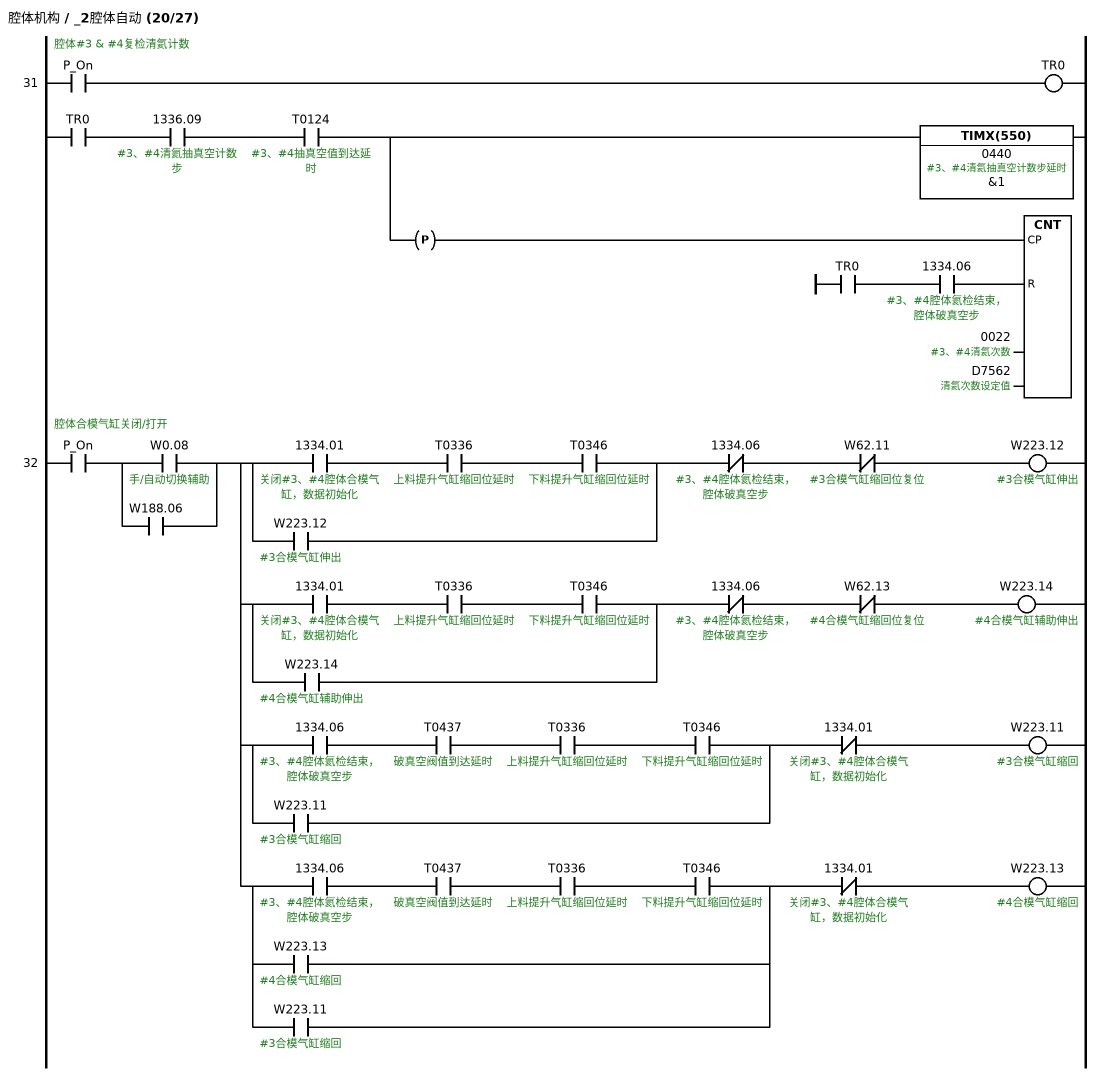
; [picture p288: 腔体机构 / _2腔体自动, rungs 31-32]
; rung 31: 腔体#3 & #4复检清氦计数
LD P_On
OUT TR0
AND 1336.09  ; #3、#4清氦抽真空计数步
AND T0124  ; #3、#4抽真空值到达延时
TIMX(550) 0440 &1  ; #3、#4清氦抽真空计数步延时
UP(521)
LD TR0
AND 1334.06  ; #3、#4腔体氦检结束，腔体破真空步
CNT 0022 D7562  ; 清氦次数设定值, #3、#4清氦次数
; rung 32: 腔体合模气缸关闭/打开
LD P_On
LD W0.08  ; 手/自动切换辅助
OR W188.06
ANDLD
OUT TR0
LD 1334.01  ; 关闭#3、#4腔体合模气缸，数据初始化
AND T0336  ; 上料提升气缸缩回位延时
AND T0346  ; 下料提升气缸缩回位延时
OR W223.12  ; #3合模气缸伸出
ANDLD
ANDNOT 1334.06  ; #3、#4腔体氦检结束，腔体破真空步
ANDNOT W62.11  ; #3合模气缸缩回位复位
OUT W223.12  ; #3合模气缸伸出
LD TR0
LD 1334.01  ; 关闭#3、#4腔体合模气缸，数据初始化
AND T0336  ; 上料提升气缸缩回位延时
AND T0346  ; 下料提升气缸缩回位延时
OR W223.14  ; #4合模气缸辅助伸出
ANDLD
ANDNOT 1334.06  ; #3、#4腔体氦检结束，腔体破真空步
ANDNOT W62.13  ; #4合模气缸缩回位复位
OUT W223.14  ; #4合模气缸辅助伸出
LD TR0
LD 1334.06  ; #3、#4腔体氦检结束，腔体破真空步
AND T0437  ; 破真空阀值到达延时
AND T0336  ; 上料提升气缸缩回位延时
AND T0346  ; 下料提升气缸缩回位延时
OR W223.11  ; #3合模气缸缩回
ANDLD
ANDNOT 1334.01  ; 关闭#3、#4腔体合模气缸，数据初始化
OUT W223.11  ; #3合模气缸缩回
LD TR0
LD 1334.06  ; #3、#4腔体氦检结束，腔体破真空步
AND T0437  ; 破真空阀值到达延时
AND T0336  ; 上料提升气缸缩回位延时
AND T0346  ; 下料提升气缸缩回位延时
LD W223.13  ; #4合模气缸缩回
OR W223.11  ; #3合模气缸缩回
ORLD
ANDLD
ANDNOT 1334.01  ; 关闭#3、#4腔体合模气缸，数据初始化
OUT W223.13  ; #4合模气缸缩回

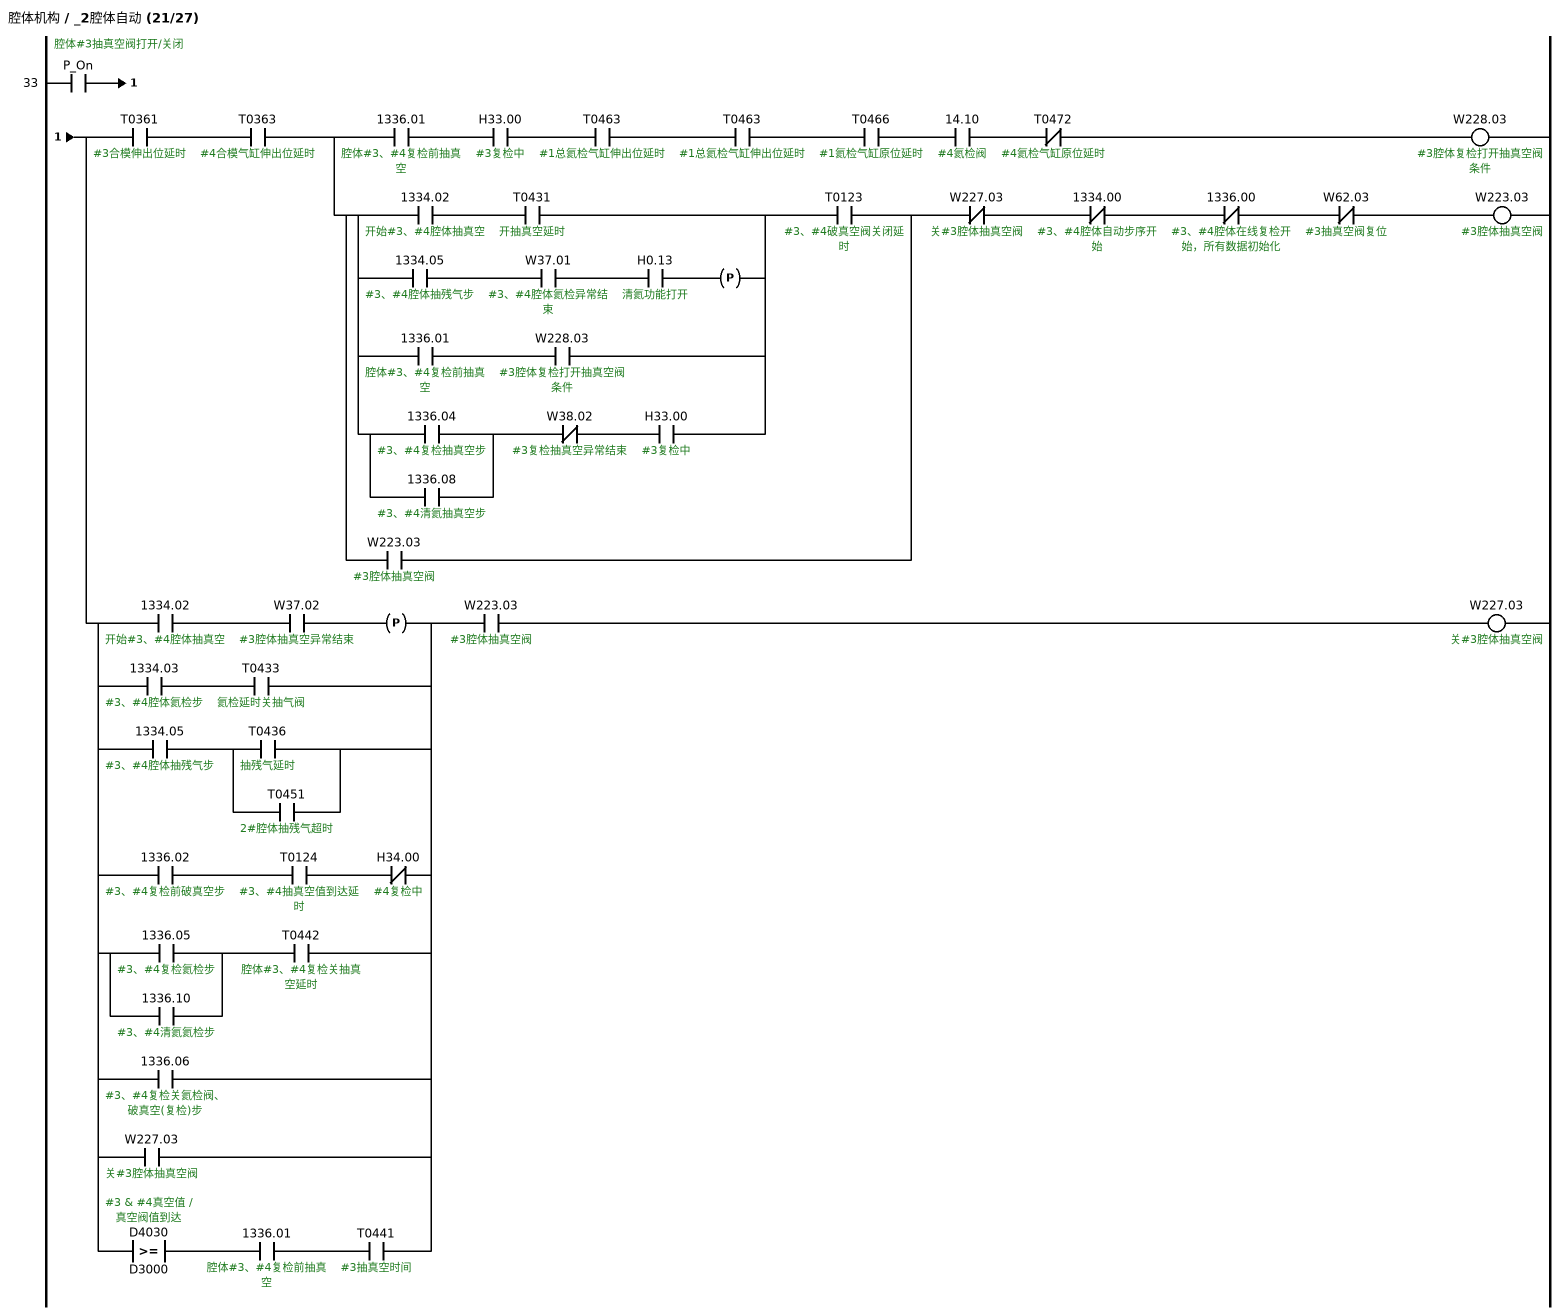
; rung 33: 腔体#3抽真空阀打开/关闭
LD P_On
OUT TR0
AND T0361  ; #3合模伸出位延时
AND T0363  ; #4合模气缸伸出位延时
OUT TR1
AND 1336.01  ; 腔体#3、#4复检前抽真空
AND H33.00  ; #3复检中
AND T0463  ; #1总氦检气缸伸出位延时
AND T0463  ; #1总氦检气缸伸出位延时
AND T0466  ; #1氦检气缸原位延时
AND 14.10  ; #4氦检阀
ANDNOT T0472  ; #4氦检气缸原位延时
OUT W228.03  ; #3腔体复检打开抽真空阀条件
LD TR1
LD 1334.02  ; 开始#3、#4腔体抽真空
AND T0431  ; 开抽真空延时
LD 1334.05  ; #3、#4腔体抽残气步
AND W37.01  ; #3、#4腔体氦检异常结束
AND H0.13  ; 清氦功能打开
UP(521)
ORLD
LD 1336.01  ; 腔体#3、#4复检前抽真空
AND W228.03  ; #3腔体复检打开抽真空阀条件
ORLD
LD 1336.04  ; #3、#4复检抽真空步
OR 1336.08  ; #3、#4清氦抽真空步
ANDNOT W38.02  ; #3复检抽真空异常结束
AND H33.00  ; #3复检中
ORLD
AND T0123  ; #3、#4破真空阀关闭延时
OR W223.03  ; #3腔体抽真空阀
ANDLD
ANDNOT W227.03  ; 关#3腔体抽真空阀
ANDNOT 1334.00  ; #3、#4腔体自动步序开始
ANDNOT 1336.00  ; #3、#4腔体在线复检开始，所有数据初始化
ANDNOT W62.03  ; #3抽真空阀复位
OUT W223.03  ; #3腔体抽真空阀
LD TR0
LD 1334.02  ; 开始#3、#4腔体抽真空
AND W37.02  ; #3腔体抽真空异常结束
UP(521)
LD 1334.03  ; #3、#4腔体氦检步
AND T0433  ; 氦检延时关抽气阀
ORLD
LD 1334.05  ; #3、#4腔体抽残气步
LD T0436  ; 抽残气延时
OR T0451  ; 2#腔体抽残气超时
ANDLD
ORLD
LD 1336.02  ; #3、#4复检前破真空步
AND T0124  ; #3、#4抽真空值到达延时
ANDNOT H34.00  ; #4复检中
ORLD
LD 1336.05  ; #3、#4复检氦检步
OR 1336.10  ; #3、#4清氦氦检步
AND T0442  ; 腔体#3、#4复检关抽真空延时
ORLD
OR 1336.06  ; #3、#4复检关氦检阀、破真空(复检)步
OR W227.03  ; 关#3腔体抽真空阀
LD>=F(334) D4030 D3000  ; #3 & #4真空值, 真空阀值到达
AND 1336.01  ; 腔体#3、#4复检前抽真空
AND T0441  ; #3抽真空时间
ORLD
ANDLD
AND W223.03  ; #3腔体抽真空阀
OUT W227.03  ; 关#3腔体抽真空阀

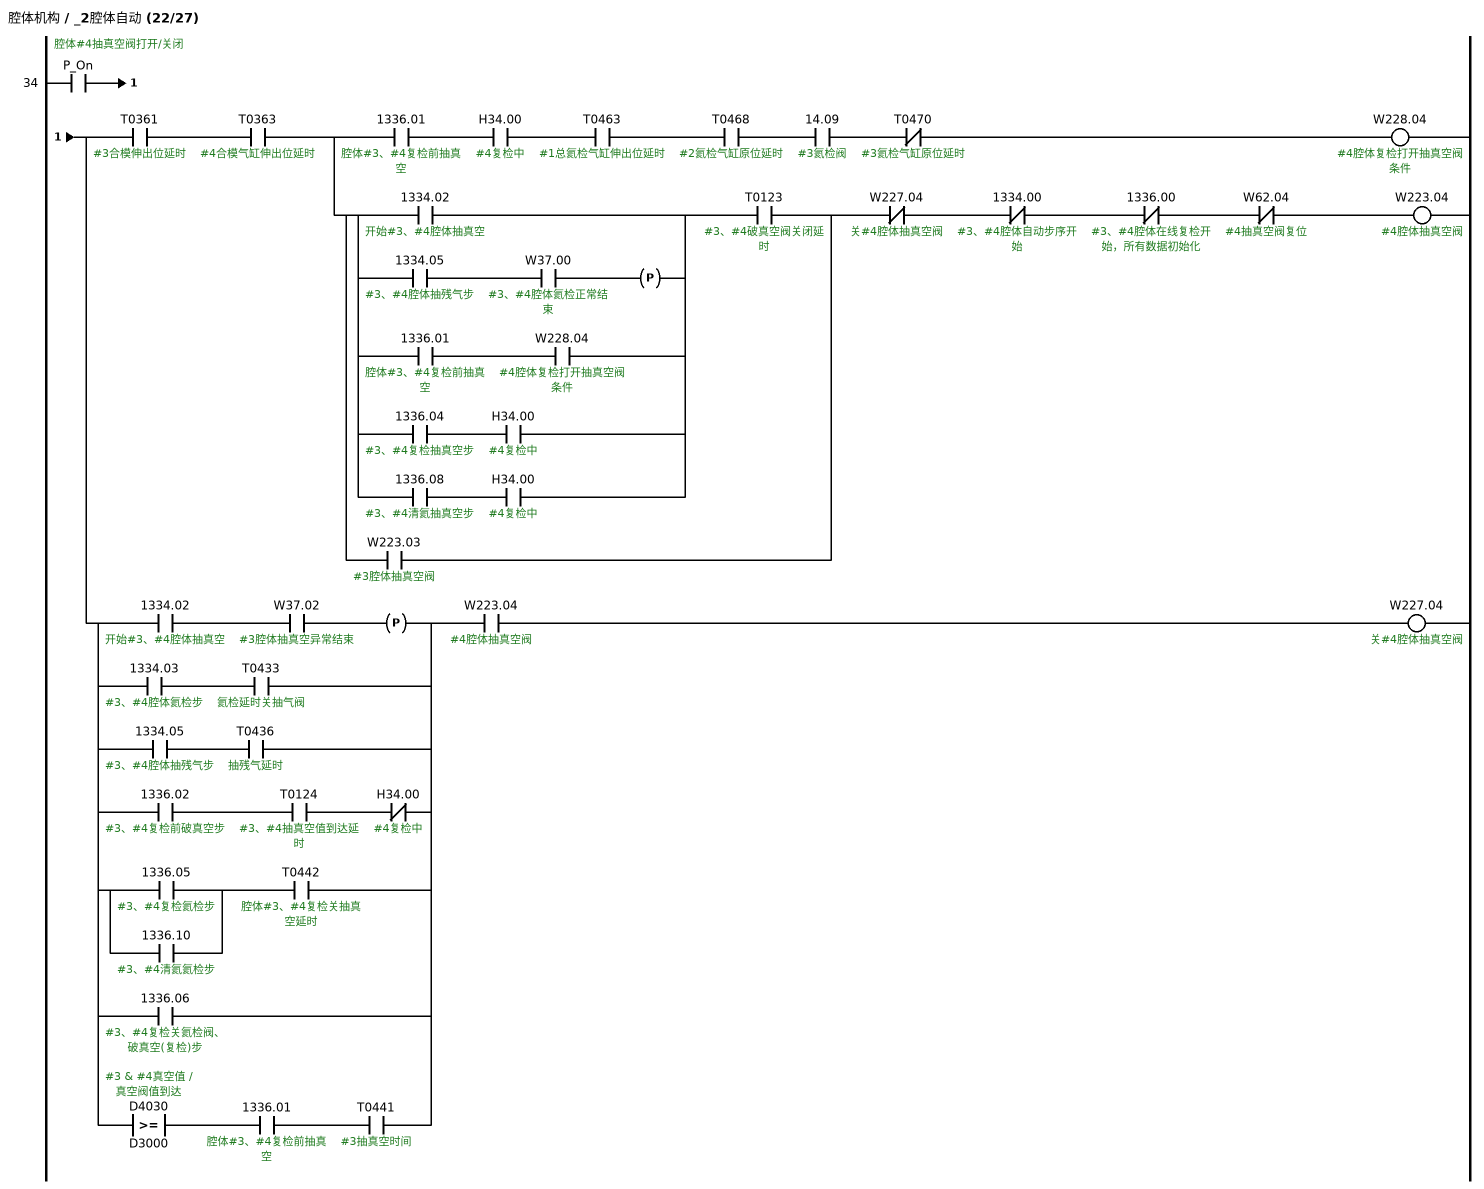
; rung 34: 腔体#4抽真空阀打开/关闭
LD P_On
OUT TR0
AND T0361  ; #3合模伸出位延时
AND T0363  ; #4合模气缸伸出位延时
OUT TR1
AND 1336.01  ; 腔体#3、#4复检前抽真空
AND H34.00  ; #4复检中
AND T0463  ; #1总氦检气缸伸出位延时
AND T0468  ; #2氦检气缸原位延时
AND 14.09  ; #3氦检阀
ANDNOT T0470  ; #3氦检气缸原位延时
OUT W228.04  ; #4腔体复检打开抽真空阀条件
LD TR1
LD 1334.02  ; 开始#3、#4腔体抽真空
LD 1334.05  ; #3、#4腔体抽残气步
AND W37.00  ; #3、#4腔体氦检正常结束
UP(521)
ORLD
LD 1336.01  ; 腔体#3、#4复检前抽真空
AND W228.04  ; #4腔体复检打开抽真空阀条件
ORLD
LD 1336.04  ; #3、#4复检抽真空步
AND H34.00  ; #4复检中
ORLD
LD 1336.08  ; #3、#4清氦抽真空步
AND H34.00  ; #4复检中
ORLD
AND T0123  ; #3、#4破真空阀关闭延时
OR W223.03  ; #3腔体抽真空阀
ANDLD
ANDNOT W227.04  ; 关#4腔体抽真空阀
ANDNOT 1334.00  ; #3、#4腔体自动步序开始
ANDNOT 1336.00  ; #3、#4腔体在线复检开始，所有数据初始化
ANDNOT W62.04  ; #4抽真空阀复位
OUT W223.04  ; #4腔体抽真空阀
LD TR0
LD 1334.02  ; 开始#3、#4腔体抽真空
AND W37.02  ; #3腔体抽真空异常结束
UP(521)
LD 1334.03  ; #3、#4腔体氦检步
AND T0433  ; 氦检延时关抽气阀
ORLD
LD 1334.05  ; #3、#4腔体抽残气步
AND T0436  ; 抽残气延时
ORLD
LD 1336.02  ; #3、#4复检前破真空步
AND T0124  ; #3、#4抽真空值到达延时
ANDNOT H34.00  ; #4复检中
ORLD
LD 1336.05  ; #3、#4复检氦检步
OR 1336.10  ; #3、#4清氦氦检步
AND T0442  ; 腔体#3、#4复检关抽真空延时
ORLD
OR 1336.06  ; #3、#4复检关氦检阀、破真空(复检)步
LD>=F(334) D4030 D3000  ; #3 & #4真空值, 真空阀值到达
AND 1336.01  ; 腔体#3、#4复检前抽真空
AND T0441  ; #3抽真空时间
ORLD
ANDLD
AND W223.04  ; #4腔体抽真空阀
OUT W227.04  ; 关#4腔体抽真空阀

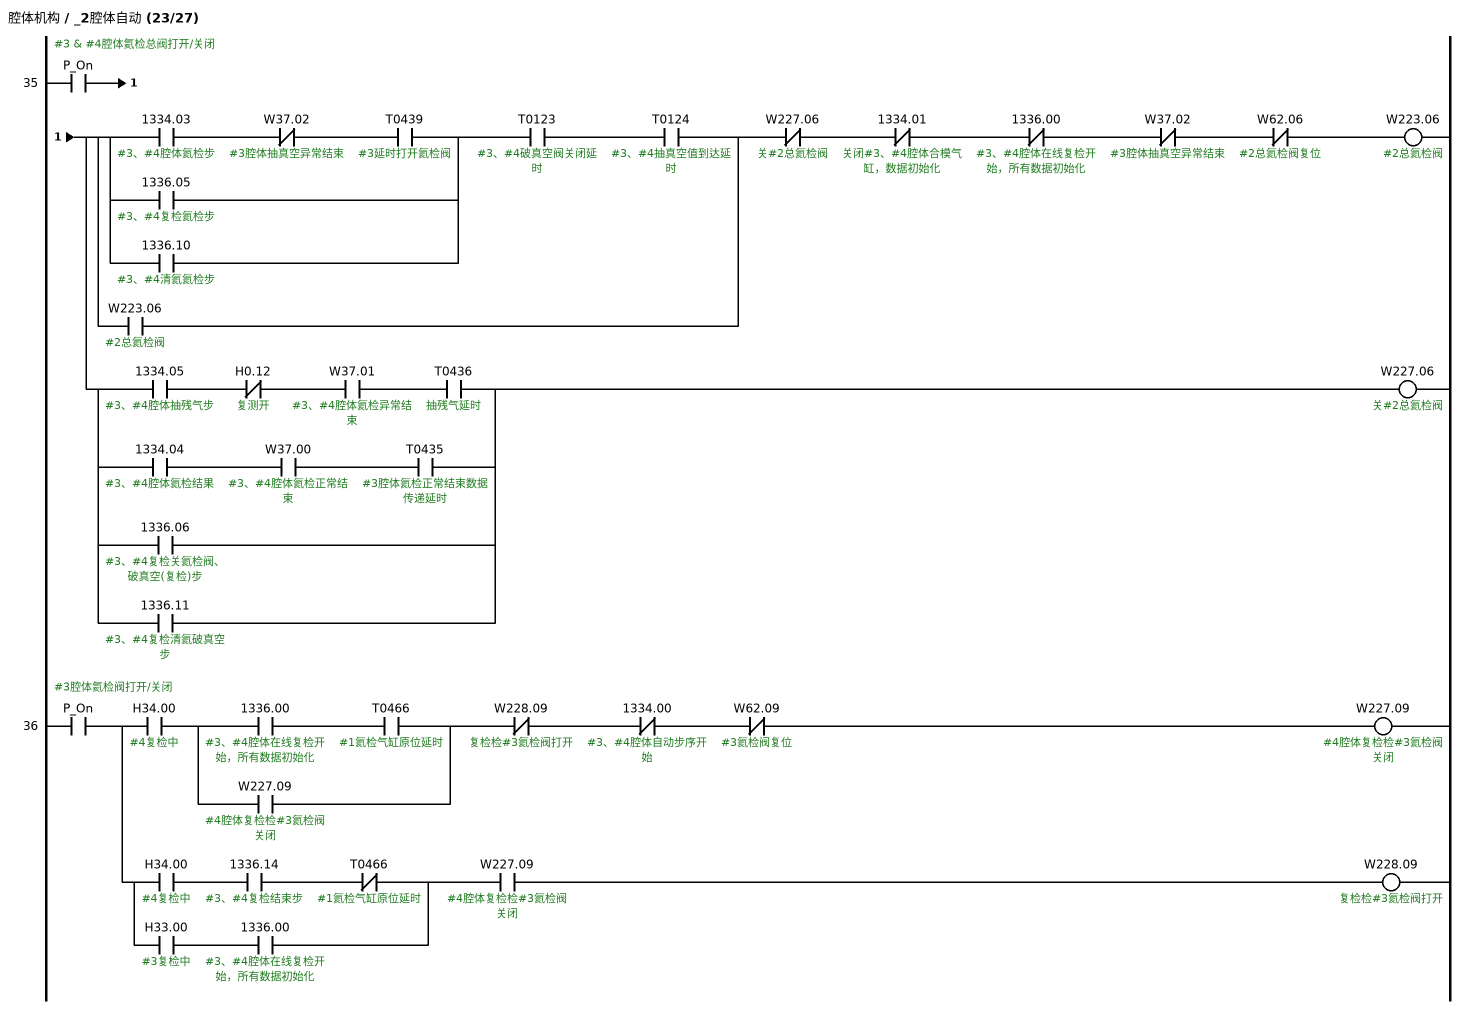
; rung 35: #3 & #4腔体氦检总阀打开/关闭
LD P_On
OUT TR0
LD 1334.03  ; #3、#4腔体氦检步
ANDNOT W37.02  ; #3腔体抽真空异常结束
AND T0439  ; #3延时打开氦检阀
OR 1336.05  ; #3、#4复检氦检步
OR 1336.10  ; #3、#4清氦氦检步
AND T0123  ; #3、#4破真空阀关闭延时
AND T0124  ; #3、#4抽真空值到达延时
OR W223.06  ; #2总氦检阀
ANDLD
ANDNOT W227.06  ; 关#2总氦检阀
ANDNOT 1334.01  ; 关闭#3、#4腔体合模气缸，数据初始化
ANDNOT 1336.00  ; #3、#4腔体在线复检开始，所有数据初始化
ANDNOT W37.02  ; #3腔体抽真空异常结束
ANDNOT W62.06  ; #2总氦检阀复位
OUT W223.06  ; #2总氦检阀
LD TR0
LD 1334.05  ; #3、#4腔体抽残气步
ANDNOT H0.12  ; 复测开
AND W37.01  ; #3、#4腔体氦检异常结束
AND T0436  ; 抽残气延时
LD 1334.04  ; #3、#4腔体氦检结果
AND W37.00  ; #3、#4腔体氦检正常结束
AND T0435  ; #3腔体氦检正常结束数据传递延时
ORLD
OR 1336.06  ; #3、#4复检关氦检阀、破真空(复检)步
OR 1336.11  ; #3、#4复检清氦破真空步
ANDLD
OUT W227.06  ; 关#2总氦检阀
; rung 36: #3腔体氦检阀打开/关闭
LD P_On
OUT TR0
AND H34.00  ; #4复检中
LD 1336.00  ; #3、#4腔体在线复检开始，所有数据初始化
AND T0466  ; #1氦检气缸原位延时
OR W227.09  ; #4腔体复检检#3氦检阀关闭
ANDLD
ANDNOT W228.09  ; 复检检#3氦检阀打开
ANDNOT 1334.00  ; #3、#4腔体自动步序开始
ANDNOT W62.09  ; #3氦检阀复位
OUT W227.09  ; #4腔体复检检#3氦检阀关闭
LD TR0
LD H34.00  ; #4复检中
AND 1336.14  ; #3、#4复检结束步
ANDNOT T0466  ; #1氦检气缸原位延时
LD H33.00  ; #3复检中
AND 1336.00  ; #3、#4腔体在线复检开始，所有数据初始化
ORLD
ANDLD
AND W227.09  ; #4腔体复检检#3氦检阀关闭
OUT W228.09  ; 复检检#3氦检阀打开

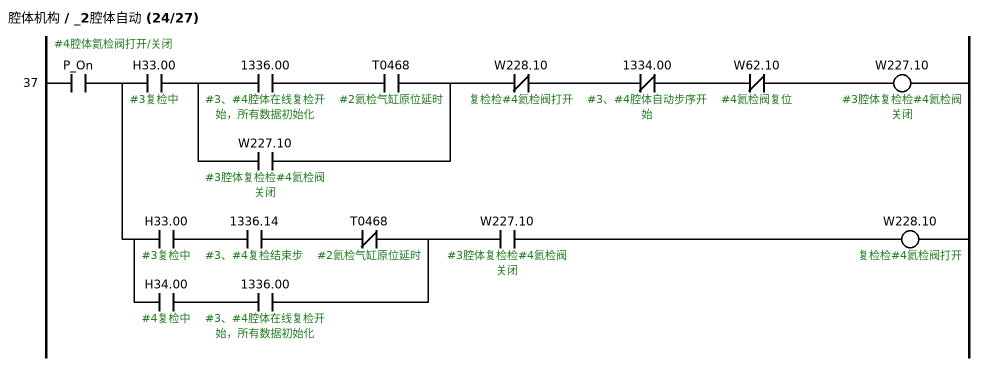
; rung 37: #4腔体氦检阀打开/关闭
LD P_On
OUT TR0
AND H33.00  ; #3复检中
LD 1336.00  ; #3、#4腔体在线复检开始，所有数据初始化
AND T0468  ; #2氦检气缸原位延时
OR W227.10  ; #3腔体复检检#4氦检阀关闭
ANDLD
ANDNOT W228.10  ; 复检检#4氦检阀打开
ANDNOT 1334.00  ; #3、#4腔体自动步序开始
ANDNOT W62.10  ; #4氦检阀复位
OUT W227.10  ; #3腔体复检检#4氦检阀关闭
LD TR0
LD H33.00  ; #3复检中
AND 1336.14  ; #3、#4复检结束步
ANDNOT T0468  ; #2氦检气缸原位延时
LD H34.00  ; #4复检中
AND 1336.00  ; #3、#4腔体在线复检开始，所有数据初始化
ORLD
ANDLD
AND W227.10  ; #3腔体复检检#4氦检阀关闭
OUT W228.10  ; 复检检#4氦检阀打开

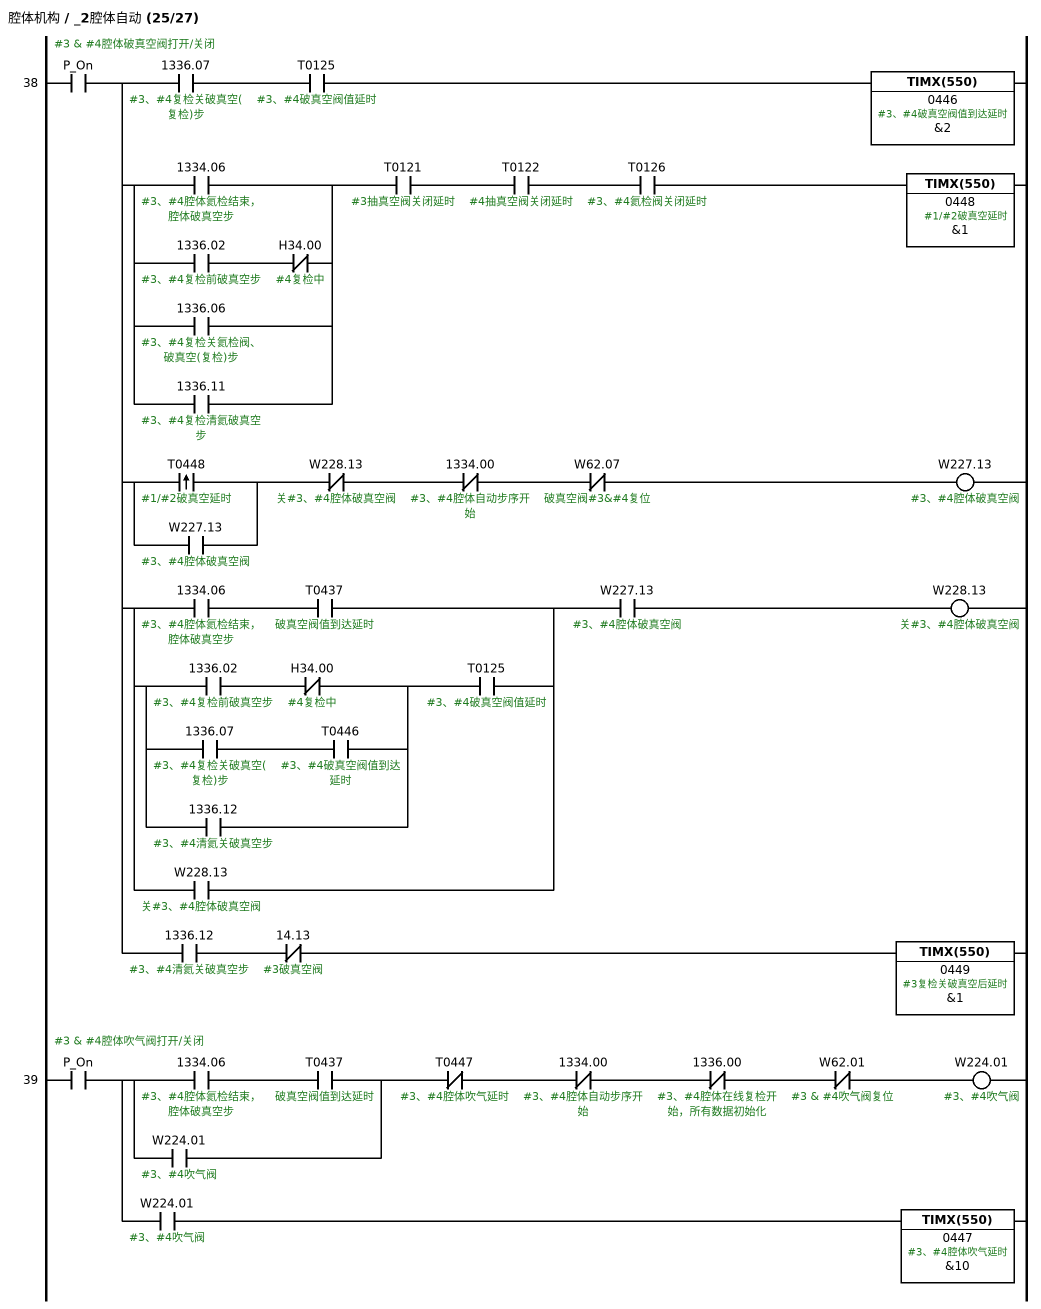
; rung 38: #3 & #4腔体破真空阀打开/关闭
LD P_On
OUT TR0
AND 1336.07  ; #3、#4复检关破真空(复检)步
AND T0125  ; #3、#4破真空阀值延时
TIMX(550) 0446 &2  ; #3、#4破真空阀值到达延时
LD TR0
LD 1334.06  ; #3、#4腔体氦检结束，腔体破真空步
LD 1336.02  ; #3、#4复检前破真空步
ANDNOT H34.00  ; #4复检中
ORLD
OR 1336.06  ; #3、#4复检关氦检阀、破真空(复检)步
OR 1336.11  ; #3、#4复检清氦破真空步
ANDLD
AND T0121  ; #3抽真空阀关闭延时
AND T0122  ; #4抽真空阀关闭延时
AND T0126  ; #3、#4氦检阀关闭延时
TIMX(550) 0448 &1  ; #1/#2破真空延时
LD TR0
@LD T0448  ; #1/#2破真空延时
OR W227.13  ; #3、#4腔体破真空阀
ANDLD
ANDNOT W228.13  ; 关#3、#4腔体破真空阀
ANDNOT 1334.00  ; #3、#4腔体自动步序开始
ANDNOT W62.07  ; 破真空阀#3&#4复位
OUT W227.13  ; #3、#4腔体破真空阀
LD TR0
LD 1334.06  ; #3、#4腔体氦检结束，腔体破真空步
AND T0437  ; 破真空阀值到达延时
LD 1336.02  ; #3、#4复检前破真空步
ANDNOT H34.00  ; #4复检中
LD 1336.07  ; #3、#4复检关破真空(复检)步
AND T0446  ; #3、#4破真空阀值到达延时
ORLD
OR 1336.12  ; #3、#4清氦关破真空步
AND T0125  ; #3、#4破真空阀值延时
ORLD
OR W228.13  ; 关#3、#4腔体破真空阀
ANDLD
AND W227.13  ; #3、#4腔体破真空阀
OUT W228.13  ; 关#3、#4腔体破真空阀
LD TR0
AND 1336.12  ; #3、#4清氦关破真空步
ANDNOT 14.13  ; #3破真空阀
TIMX(550) 0449 &1  ; #3复检关破真空后延时
; rung 39: #3 & #4腔体吹气阀打开/关闭
LD P_On
OUT TR0
LD 1334.06  ; #3、#4腔体氦检结束，腔体破真空步
AND T0437  ; 破真空阀值到达延时
OR W224.01  ; #3、#4吹气阀
ANDLD
ANDNOT T0447  ; #3、#4腔体吹气延时
ANDNOT 1334.00  ; #3、#4腔体自动步序开始
ANDNOT 1336.00  ; #3、#4腔体在线复检开始，所有数据初始化
ANDNOT W62.01  ; #3 & #4吹气阀复位
OUT W224.01  ; #3、#4吹气阀
LD TR0
AND W224.01  ; #3、#4吹气阀
TIMX(550) 0447 &10  ; #3、#4腔体吹气延时

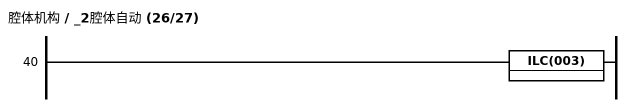
; rung 40
ILC(003)

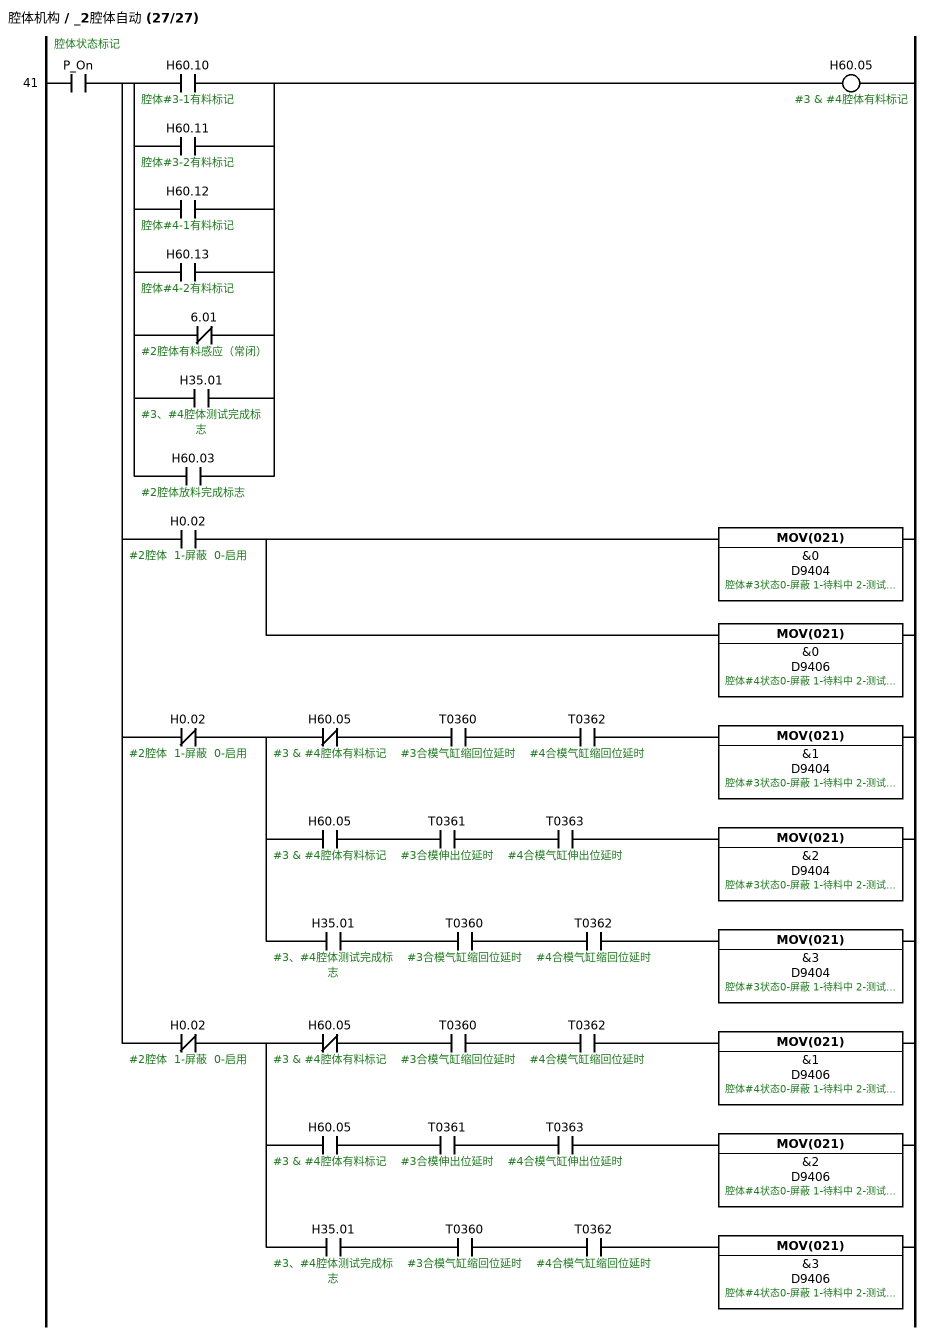
; rung 41: 腔体状态标记
LD P_On
OUT TR0
LD H60.10  ; 腔体#3-1有料标记
OR H60.11  ; 腔体#3-2有料标记
OR H60.12  ; 腔体#4-1有料标记
OR H60.13  ; 腔体#4-2有料标记
ORNOT 6.01  ; #2腔体有料感应（常闭）
OR H35.01  ; #3、#4腔体测试完成标志
OR H60.03  ; #2腔体放料完成标志
ANDLD
OUT H60.05  ; #3 & #4腔体有料标记
LD TR0
AND H0.02  ; #2腔体  1-屏蔽  0-启用
MOV(021) &0 D9404  ; 腔体#3状态0-屏蔽 1-待料中 2-测试中 3-测试完成 4-在线复检
MOV(021) &0 D9406  ; 腔体#4状态0-屏蔽 1-待料中 2-测试中 3-测试完成 4-在线复检
LD TR0
ANDNOT H0.02  ; #2腔体  1-屏蔽  0-启用
OUT TR1
ANDNOT H60.05  ; #3 & #4腔体有料标记
AND T0360  ; #3合模气缸缩回位延时
AND T0362  ; #4合模气缸缩回位延时
MOV(021) &1 D9404  ; 腔体#3状态0-屏蔽 1-待料中 2-测试中 3-测试完成 4-在线复检
LD TR1
AND H60.05  ; #3 & #4腔体有料标记
AND T0361  ; #3合模伸出位延时
AND T0363  ; #4合模气缸伸出位延时
MOV(021) &2 D9404  ; 腔体#3状态0-屏蔽 1-待料中 2-测试中 3-测试完成 4-在线复检
LD TR1
AND H35.01  ; #3、#4腔体测试完成标志
AND T0360  ; #3合模气缸缩回位延时
AND T0362  ; #4合模气缸缩回位延时
MOV(021) &3 D9404  ; 腔体#3状态0-屏蔽 1-待料中 2-测试中 3-测试完成 4-在线复检
LD TR0
ANDNOT H0.02  ; #2腔体  1-屏蔽  0-启用
OUT TR0
ANDNOT H60.05  ; #3 & #4腔体有料标记
AND T0360  ; #3合模气缸缩回位延时
AND T0362  ; #4合模气缸缩回位延时
MOV(021) &1 D9406  ; 腔体#4状态0-屏蔽 1-待料中 2-测试中 3-测试完成 4-在线复检
LD TR0
AND H60.05  ; #3 & #4腔体有料标记
AND T0361  ; #3合模伸出位延时
AND T0363  ; #4合模气缸伸出位延时
MOV(021) &2 D9406  ; 腔体#4状态0-屏蔽 1-待料中 2-测试中 3-测试完成 4-在线复检
LD TR0
AND H35.01  ; #3、#4腔体测试完成标志
AND T0360  ; #3合模气缸缩回位延时
AND T0362  ; #4合模气缸缩回位延时
MOV(021) &3 D9406  ; 腔体#4状态0-屏蔽 1-待料中 2-测试中 3-测试完成 4-在线复检

### Section 腔体机构手动

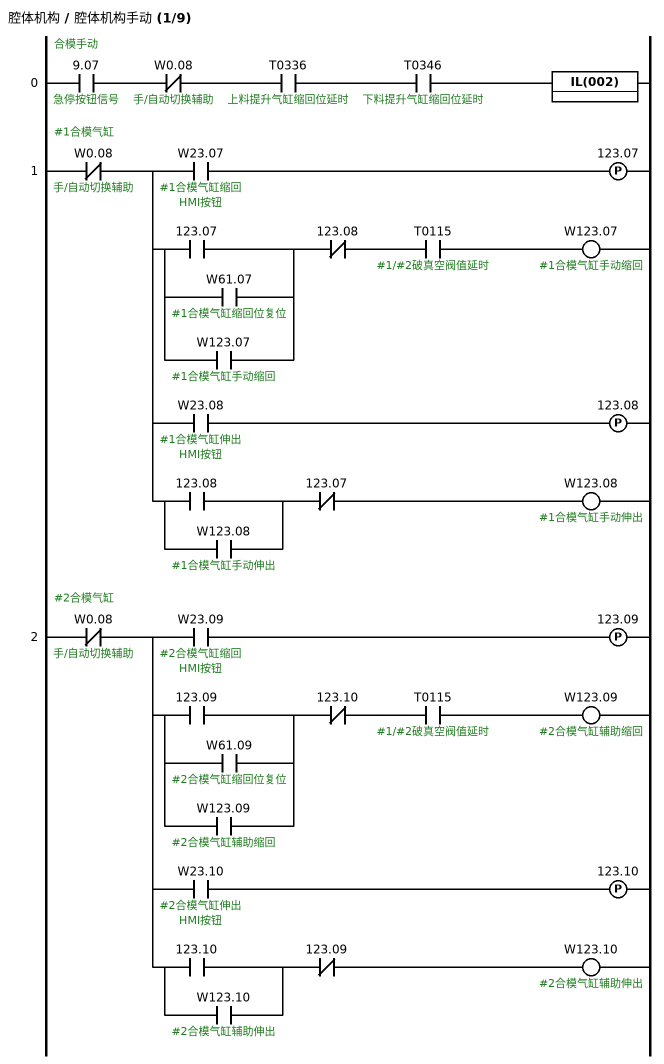
; rung 0: 合模手动
LD 9.07  ; 急停按钮信号
ANDNOT W0.08  ; 手/自动切换辅助
AND T0336  ; 上料提升气缸缩回位延时
AND T0346  ; 下料提升气缸缩回位延时
IL(002)
; rung 1: #1合模气缸
LDNOT W0.08  ; 手/自动切换辅助
OUT TR0
AND W23.07  ; #1合模气缸缩回   HMI按钮
DIFU(013) 123.07
LD TR0
LD 123.07
OR W61.07  ; #1合模气缸缩回位复位
OR W123.07  ; #1合模气缸手动缩回
ANDLD
ANDNOT 123.08
AND T0115  ; #1/#2破真空阀值延时
OUT W123.07  ; #1合模气缸手动缩回
LD TR0
AND W23.08  ; #1合模气缸伸出   HMI按钮
DIFU(013) 123.08
LD TR0
LD 123.08
OR W123.08  ; #1合模气缸手动伸出
ANDLD
ANDNOT 123.07
OUT W123.08  ; #1合模气缸手动伸出
; rung 2: #2合模气缸
LDNOT W0.08  ; 手/自动切换辅助
OUT TR0
AND W23.09  ; #2合模气缸缩回   HMI按钮
DIFU(013) 123.09
LD TR0
LD 123.09
OR W61.09  ; #2合模气缸缩回位复位
OR W123.09  ; #2合模气缸辅助缩回
ANDLD
ANDNOT 123.10
AND T0115  ; #1/#2破真空阀值延时
OUT W123.09  ; #2合模气缸辅助缩回
LD TR0
AND W23.10  ; #2合模气缸伸出   HMI按钮
DIFU(013) 123.10
LD TR0
LD 123.10
OR W123.10  ; #2合模气缸辅助伸出
ANDLD
ANDNOT 123.09
OUT W123.10  ; #2合模气缸辅助伸出

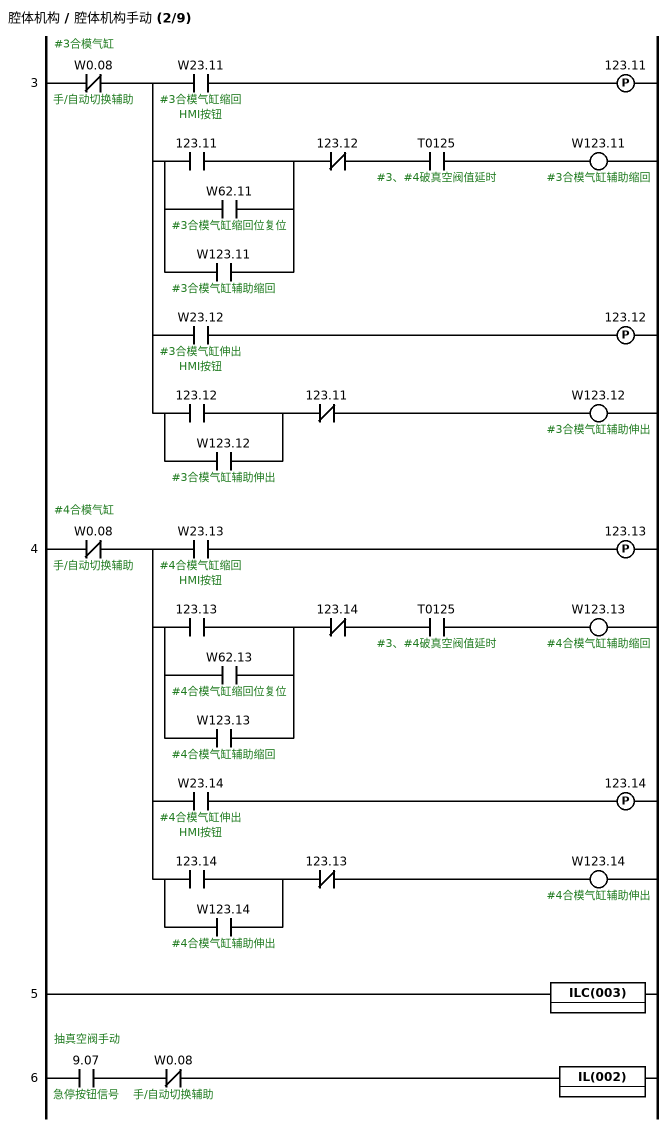
; rung 3: #3合模气缸
LDNOT W0.08  ; 手/自动切换辅助
OUT TR0
AND W23.11  ; #3合模气缸缩回   HMI按钮
DIFU(013) 123.11
LD TR0
LD 123.11
OR W62.11  ; #3合模气缸缩回位复位
OR W123.11  ; #3合模气缸辅助缩回
ANDLD
ANDNOT 123.12
AND T0125  ; #3、#4破真空阀值延时
OUT W123.11  ; #3合模气缸辅助缩回
LD TR0
AND W23.12  ; #3合模气缸伸出   HMI按钮
DIFU(013) 123.12
LD TR0
LD 123.12
OR W123.12  ; #3合模气缸辅助伸出
ANDLD
ANDNOT 123.11
OUT W123.12  ; #3合模气缸辅助伸出
; rung 4: #4合模气缸
LDNOT W0.08  ; 手/自动切换辅助
OUT TR0
AND W23.13  ; #4合模气缸缩回   HMI按钮
DIFU(013) 123.13
LD TR0
LD 123.13
OR W62.13  ; #4合模气缸缩回位复位
OR W123.13  ; #4合模气缸辅助缩回
ANDLD
ANDNOT 123.14
AND T0125  ; #3、#4破真空阀值延时
OUT W123.13  ; #4合模气缸辅助缩回
LD TR0
AND W23.14  ; #4合模气缸伸出   HMI按钮
DIFU(013) 123.14
LD TR0
LD 123.14
OR W123.14  ; #4合模气缸辅助伸出
ANDLD
ANDNOT 123.13
OUT W123.14  ; #4合模气缸辅助伸出
; rung 5
ILC(003)
; rung 6: 抽真空阀手动
LD 9.07  ; 急停按钮信号
ANDNOT W0.08  ; 手/自动切换辅助
IL(002)

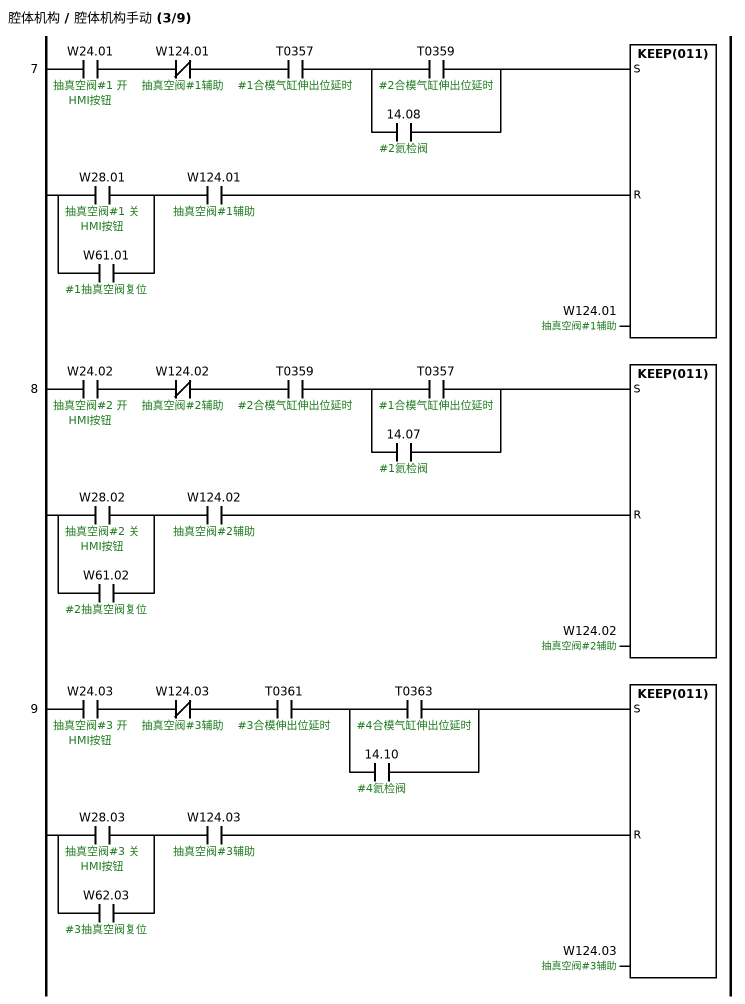
; rung 7
LD W24.01  ; 抽真空阀#1 开    HMI按钮
ANDNOT W124.01  ; 抽真空阀#1辅助
AND T0357  ; #1合模气缸伸出位延时
LD T0359  ; #2合模气缸伸出位延时
OR 14.08  ; #2氦检阀
ANDLD
LD W28.01  ; 抽真空阀#1 关    HMI按钮
OR W61.01  ; #1抽真空阀复位
AND W124.01  ; 抽真空阀#1辅助
KEEP(011) W124.01  ; 抽真空阀#1辅助
; rung 8
LD W24.02  ; 抽真空阀#2 开    HMI按钮
ANDNOT W124.02  ; 抽真空阀#2辅助
AND T0359  ; #2合模气缸伸出位延时
LD T0357  ; #1合模气缸伸出位延时
OR 14.07  ; #1氦检阀
ANDLD
LD W28.02  ; 抽真空阀#2 关    HMI按钮
OR W61.02  ; #2抽真空阀复位
AND W124.02  ; 抽真空阀#2辅助
KEEP(011) W124.02  ; 抽真空阀#2辅助
; rung 9
LD W24.03  ; 抽真空阀#3 开    HMI按钮
ANDNOT W124.03  ; 抽真空阀#3辅助
AND T0361  ; #3合模伸出位延时
LD T0363  ; #4合模气缸伸出位延时
OR 14.10  ; #4氦检阀
ANDLD
LD W28.03  ; 抽真空阀#3 关    HMI按钮
OR W62.03  ; #3抽真空阀复位
AND W124.03  ; 抽真空阀#3辅助
KEEP(011) W124.03  ; 抽真空阀#3辅助

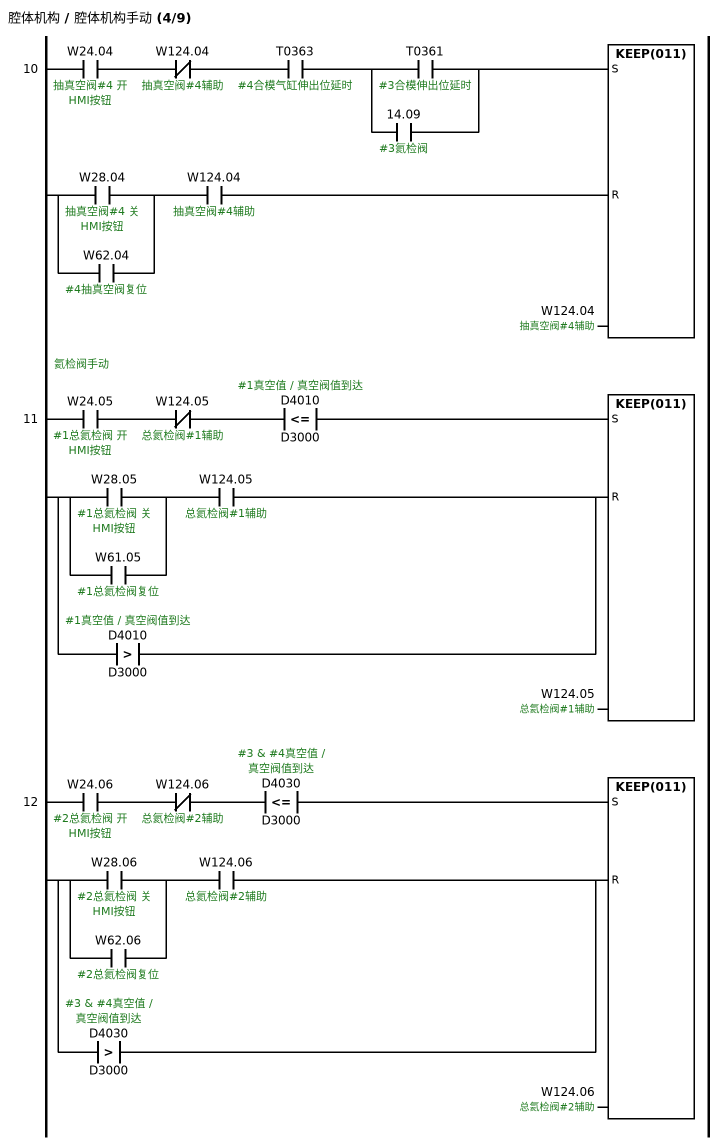
; rung 10
LD W24.04  ; 抽真空阀#4 开    HMI按钮
ANDNOT W124.04  ; 抽真空阀#4辅助
AND T0363  ; #4合模气缸伸出位延时
LD T0361  ; #3合模伸出位延时
OR 14.09  ; #3氦检阀
ANDLD
LD W28.04  ; 抽真空阀#4 关    HMI按钮
OR W62.04  ; #4抽真空阀复位
AND W124.04  ; 抽真空阀#4辅助
KEEP(011) W124.04  ; 抽真空阀#4辅助
; rung 11: 氦检阀手动
LD W24.05  ; #1总氦检阀 开    HMI按钮
ANDNOT W124.05  ; 总氦检阀#1辅助
AND<=F(332) D4010 D3000  ; #1真空值, 真空阀值到达
LD W28.05  ; #1总氦检阀 关    HMI按钮
OR W61.05  ; #1总氦检阀复位
AND W124.05  ; 总氦检阀#1辅助
OR>F(333) D4010 D3000  ; #1真空值, 真空阀值到达
KEEP(011) W124.05  ; 总氦检阀#1辅助
; rung 12
LD W24.06  ; #2总氦检阀 开    HMI按钮
ANDNOT W124.06  ; 总氦检阀#2辅助
AND<=F(332) D4030 D3000  ; #3 & #4真空值, 真空阀值到达
LD W28.06  ; #2总氦检阀 关    HMI按钮
OR W62.06  ; #2总氦检阀复位
AND W124.06  ; 总氦检阀#2辅助
OR>F(333) D4030 D3000  ; #3 & #4真空值, 真空阀值到达
KEEP(011) W124.06  ; 总氦检阀#2辅助

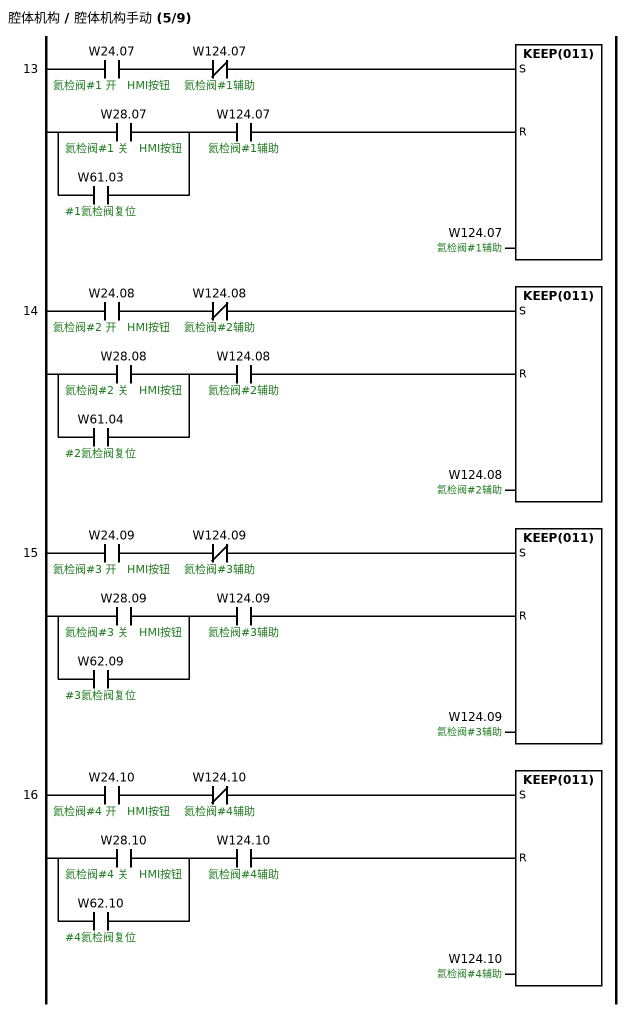
; rung 13
LD W24.07  ; 氦检阀#1 开   HMI按钮
ANDNOT W124.07  ; 氦检阀#1辅助
LD W28.07  ; 氦检阀#1 关   HMI按钮
OR W61.03  ; #1氦检阀复位
AND W124.07  ; 氦检阀#1辅助
KEEP(011) W124.07  ; 氦检阀#1辅助
; rung 14
LD W24.08  ; 氦检阀#2 开   HMI按钮
ANDNOT W124.08  ; 氦检阀#2辅助
LD W28.08  ; 氦检阀#2 关   HMI按钮
OR W61.04  ; #2氦检阀复位
AND W124.08  ; 氦检阀#2辅助
KEEP(011) W124.08  ; 氦检阀#2辅助
; rung 15
LD W24.09  ; 氦检阀#3 开   HMI按钮
ANDNOT W124.09  ; 氦检阀#3辅助
LD W28.09  ; 氦检阀#3 关   HMI按钮
OR W62.09  ; #3氦检阀复位
AND W124.09  ; 氦检阀#3辅助
KEEP(011) W124.09  ; 氦检阀#3辅助
; rung 16
LD W24.10  ; 氦检阀#4 开   HMI按钮
ANDNOT W124.10  ; 氦检阀#4辅助
LD W28.10  ; 氦检阀#4 关   HMI按钮
OR W62.10  ; #4氦检阀复位
AND W124.10  ; 氦检阀#4辅助
KEEP(011) W124.10  ; 氦检阀#4辅助

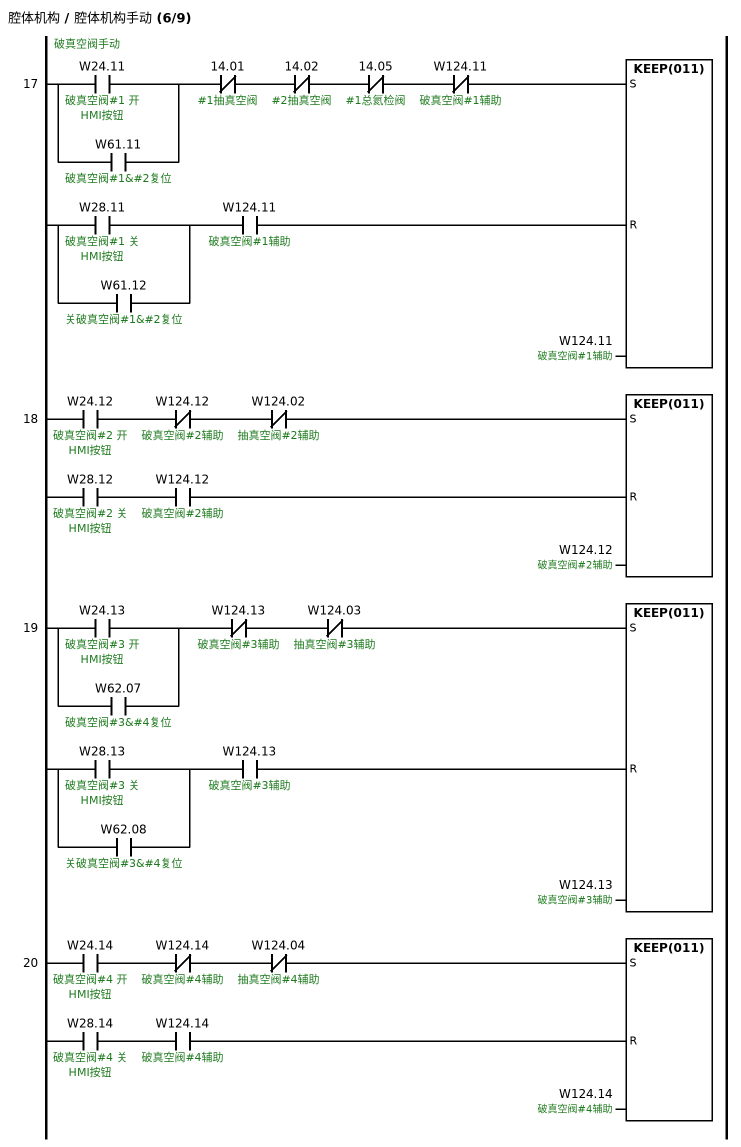
; rung 17: 破真空阀手动
LD W24.11  ; 破真空阀#1 开   HMI按钮
OR W61.11  ; 破真空阀#1&#2复位
ANDNOT 14.01  ; #1抽真空阀
ANDNOT 14.02  ; #2抽真空阀
ANDNOT 14.05  ; #1总氦检阀
ANDNOT W124.11  ; 破真空阀#1辅助
LD W28.11  ; 破真空阀#1 关   HMI按钮
OR W61.12  ; 关破真空阀#1&#2复位
AND W124.11  ; 破真空阀#1辅助
KEEP(011) W124.11  ; 破真空阀#1辅助
; rung 18
LD W24.12  ; 破真空阀#2 开   HMI按钮
ANDNOT W124.12  ; 破真空阀#2辅助
ANDNOT W124.02  ; 抽真空阀#2辅助
LD W28.12  ; 破真空阀#2 关   HMI按钮
AND W124.12  ; 破真空阀#2辅助
KEEP(011) W124.12  ; 破真空阀#2辅助
; rung 19
LD W24.13  ; 破真空阀#3 开   HMI按钮
OR W62.07  ; 破真空阀#3&#4复位
ANDNOT W124.13  ; 破真空阀#3辅助
ANDNOT W124.03  ; 抽真空阀#3辅助
LD W28.13  ; 破真空阀#3 关   HMI按钮
OR W62.08  ; 关破真空阀#3&#4复位
AND W124.13  ; 破真空阀#3辅助
KEEP(011) W124.13  ; 破真空阀#3辅助
; rung 20
LD W24.14  ; 破真空阀#4 开   HMI按钮
ANDNOT W124.14  ; 破真空阀#4辅助
ANDNOT W124.04  ; 抽真空阀#4辅助
LD W28.14  ; 破真空阀#4 关   HMI按钮
AND W124.14  ; 破真空阀#4辅助
KEEP(011) W124.14  ; 破真空阀#4辅助

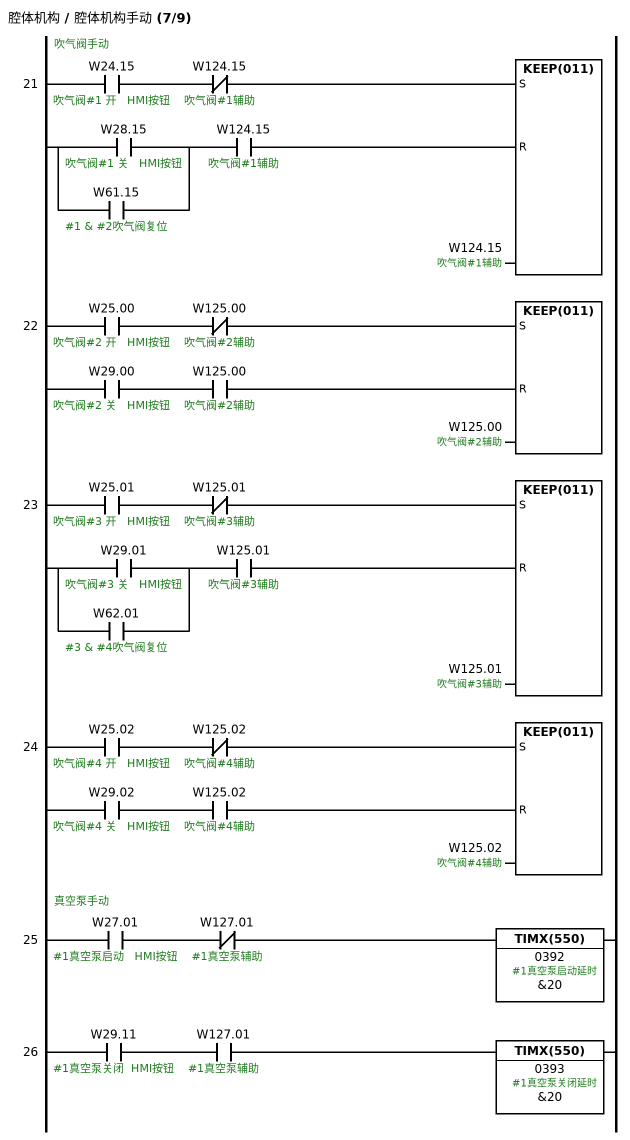
; rung 21: 吹气阀手动
LD W24.15  ; 吹气阀#1 开   HMI按钮
ANDNOT W124.15  ; 吹气阀#1辅助
LD W28.15  ; 吹气阀#1 关   HMI按钮
OR W61.15  ; #1 & #2吹气阀复位
AND W124.15  ; 吹气阀#1辅助
KEEP(011) W124.15  ; 吹气阀#1辅助
; rung 22
LD W25.00  ; 吹气阀#2 开   HMI按钮
ANDNOT W125.00  ; 吹气阀#2辅助
LD W29.00  ; 吹气阀#2 关   HMI按钮
AND W125.00  ; 吹气阀#2辅助
KEEP(011) W125.00  ; 吹气阀#2辅助
; rung 23
LD W25.01  ; 吹气阀#3 开   HMI按钮
ANDNOT W125.01  ; 吹气阀#3辅助
LD W29.01  ; 吹气阀#3 关   HMI按钮
OR W62.01  ; #3 & #4吹气阀复位
AND W125.01  ; 吹气阀#3辅助
KEEP(011) W125.01  ; 吹气阀#3辅助
; rung 24
LD W25.02  ; 吹气阀#4 开   HMI按钮
ANDNOT W125.02  ; 吹气阀#4辅助
LD W29.02  ; 吹气阀#4 关   HMI按钮
AND W125.02  ; 吹气阀#4辅助
KEEP(011) W125.02  ; 吹气阀#4辅助
; rung 25: 真空泵手动
LD W27.01  ; #1真空泵启动   HMI按钮
ANDNOT W127.01  ; #1真空泵辅助
TIMX(550) 0392 &20  ; #1真空泵启动延时
; rung 26
LD W29.11  ; #1真空泵关闭  HMI按钮
AND W127.01  ; #1真空泵辅助
TIMX(550) 0393 &20  ; #1真空泵关闭延时

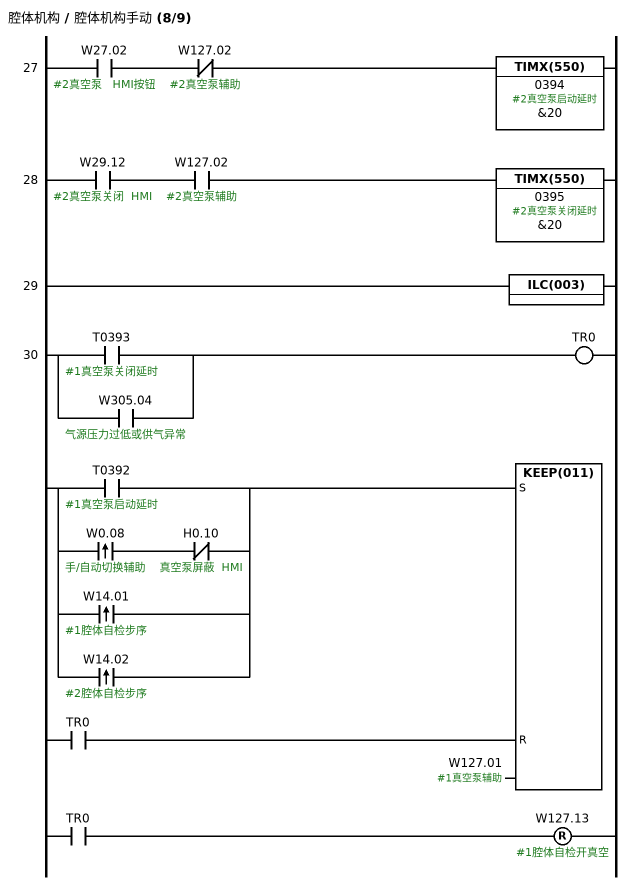
; rung 27
LD W27.02  ; #2真空泵   HMI按钮
ANDNOT W127.02  ; #2真空泵辅助
TIMX(550) 0394 &20  ; #2真空泵启动延时
; rung 28
LD W29.12  ; #2真空泵关闭  HMI
AND W127.02  ; #2真空泵辅助
TIMX(550) 0395 &20  ; #2真空泵关闭延时
; rung 29
ILC(003)
; rung 30
LD T0392  ; #1真空泵启动延时
@LD W0.08  ; 手/自动切换辅助
ANDNOT H0.10  ; 真空泵屏蔽  HMI
ORLD
@OR W14.01  ; #1腔体自检步序
@OR W14.02  ; #2腔体自检步序
LD T0393  ; #1真空泵关闭延时
OR W305.04  ; 气源压力过低或供气异常
OUT TR0
KEEP(011) W127.01  ; #1真空泵辅助
LD TR0
RSET W127.13  ; #1腔体自检开真空

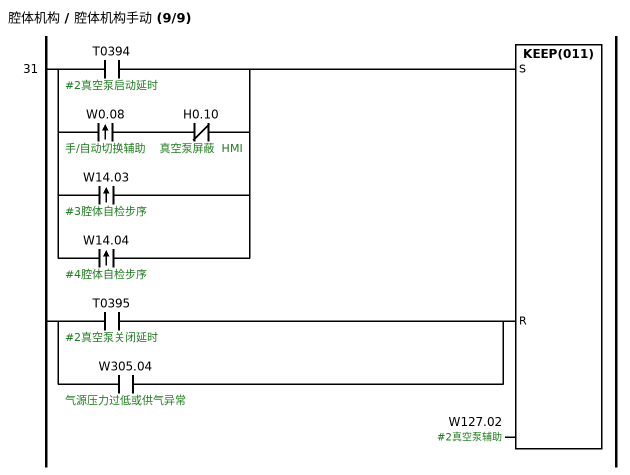
; rung 31
LD T0394  ; #2真空泵启动延时
@LD W0.08  ; 手/自动切换辅助
ANDNOT H0.10  ; 真空泵屏蔽  HMI
ORLD
@OR W14.03  ; #3腔体自检步序
@OR W14.04  ; #4腔体自检步序
LD T0395  ; #2真空泵关闭延时
OR W305.04  ; 气源压力过低或供气异常
KEEP(011) W127.02  ; #2真空泵辅助

### Section _1腔体自检

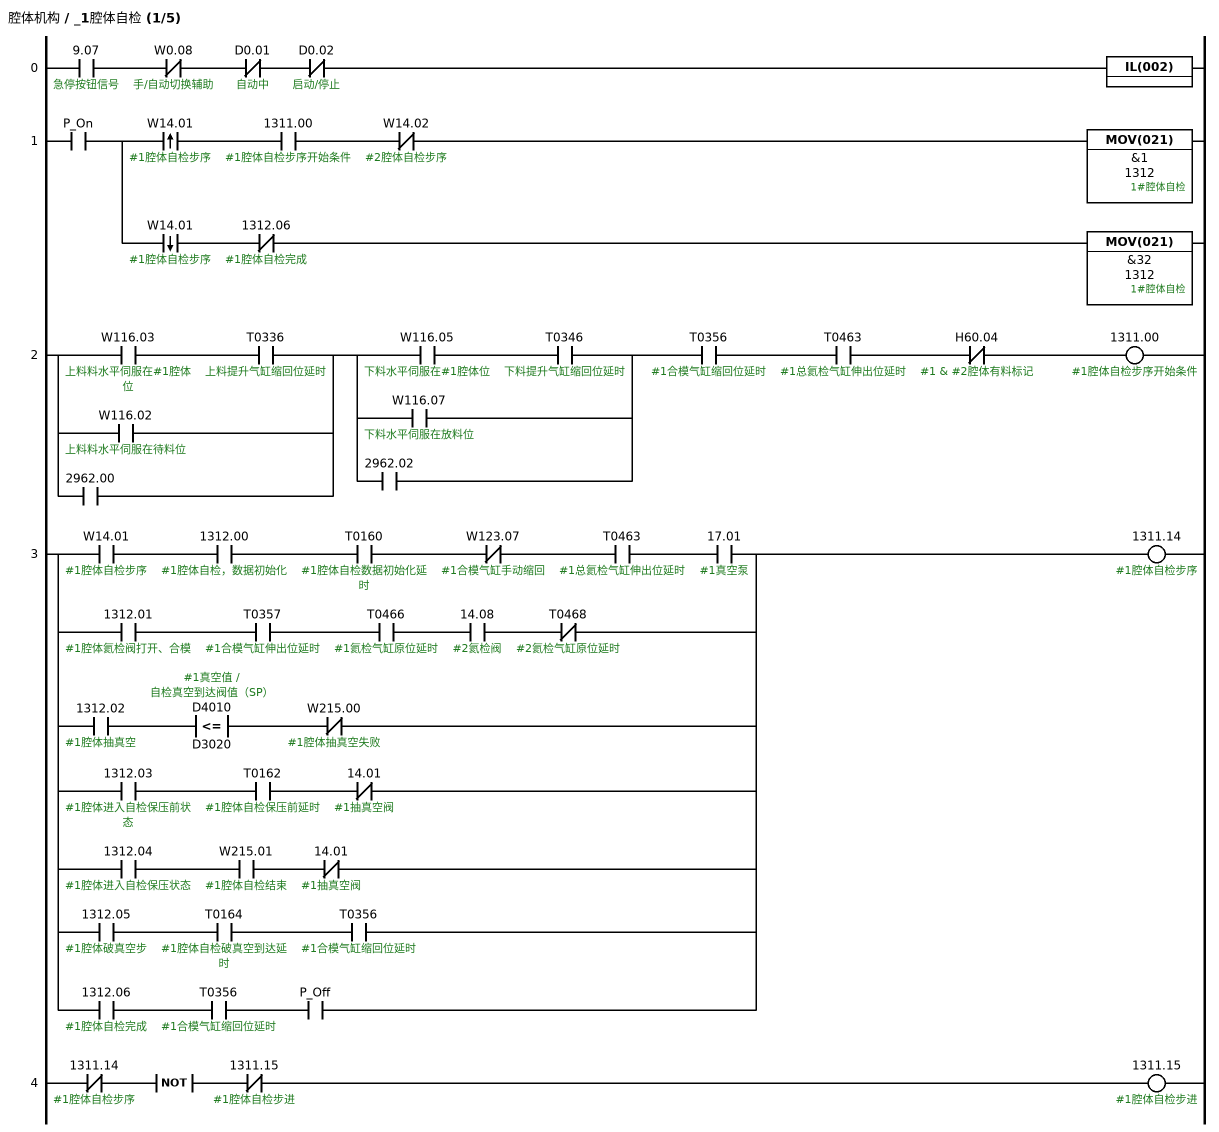
; rung 0
LD 9.07  ; 急停按钮信号
ANDNOT W0.08  ; 手/自动切换辅助
ANDNOT D0.01  ; 自动中
ANDNOT D0.02  ; 启动/停止
IL(002)
; rung 1
LD P_On
OUT TR0
@AND W14.01  ; #1腔体自检步序
AND 1311.00  ; #1腔体自检步序开始条件
ANDNOT W14.02  ; #2腔体自检步序
MOV(021) &1 1312  ; 1#腔体自检
LD TR0
%AND W14.01  ; #1腔体自检步序
ANDNOT 1312.06  ; #1腔体自检完成
MOV(021) &32 1312  ; 1#腔体自检
; rung 2
LD W116.03  ; 上料料水平伺服在#1腔体位
AND T0336  ; 上料提升气缸缩回位延时
OR W116.02  ; 上料料水平伺服在待料位
OR 2962.00
LD W116.05  ; 下料水平伺服在#1腔体位
AND T0346  ; 下料提升气缸缩回位延时
OR W116.07  ; 下料水平伺服在放料位
OR 2962.02
ANDLD
AND T0356  ; #1合模气缸缩回位延时
AND T0463  ; #1总氦检气缸伸出位延时
ANDNOT H60.04  ; #1 & #2腔体有料标记
OUT 1311.00  ; #1腔体自检步序开始条件
; rung 3
LD W14.01  ; #1腔体自检步序
AND 1312.00  ; #1腔体自检，数据初始化
AND T0160  ; #1腔体自检数据初始化延时
ANDNOT W123.07  ; #1合模气缸手动缩回
AND T0463  ; #1总氦检气缸伸出位延时
AND 17.01  ; #1真空泵
LD 1312.01  ; #1腔体氦检阀打开、合模
AND T0357  ; #1合模气缸伸出位延时
AND T0466  ; #1氦检气缸原位延时
AND 14.08  ; #2氦检阀
ANDNOT T0468  ; #2氦检气缸原位延时
ORLD
LD 1312.02  ; #1腔体抽真空
AND<=F(332) D4010 D3020  ; #1真空值, 自检真空到达阀值（SP）
ANDNOT W215.00  ; #1腔体抽真空失败
ORLD
LD 1312.03  ; #1腔体进入自检保压前状态
AND T0162  ; #1腔体自检保压前延时
ANDNOT 14.01  ; #1抽真空阀
ORLD
LD 1312.04  ; #1腔体进入自检保压状态
AND W215.01  ; #1腔体自检结束
ANDNOT 14.01  ; #1抽真空阀
ORLD
LD 1312.05  ; #1腔体破真空步
AND T0164  ; #1腔体自检破真空到达延时
AND T0356  ; #1合模气缸缩回位延时
ORLD
LD 1312.06  ; #1腔体自检完成
AND T0356  ; #1合模气缸缩回位延时
AND P_Off
ORLD
OUT 1311.14  ; #1腔体自检步序
; rung 4
LDNOT 1311.14  ; #1腔体自检步序
NOT(520)
ANDNOT 1311.15  ; #1腔体自检步进
OUT 1311.15  ; #1腔体自检步进

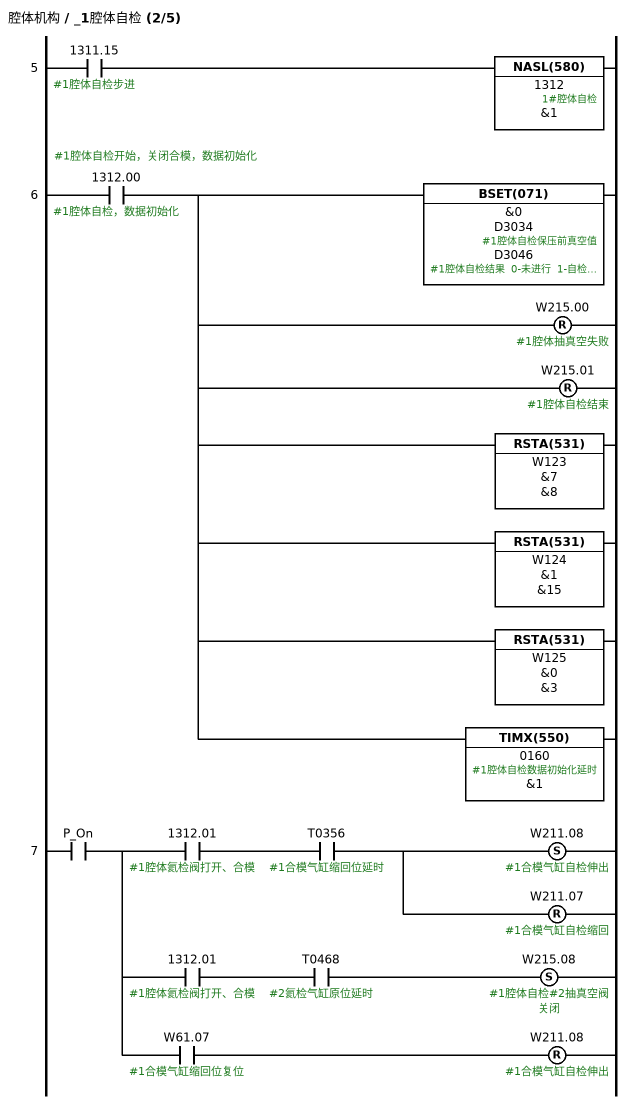
; rung 5
LD 1311.15  ; #1腔体自检步进
NASL(580) 1312 &1  ; 1#腔体自检
; rung 6: #1腔体自检开始，关闭合模，数据初始化
LD 1312.00  ; #1腔体自检，数据初始化
BSET(071) &0 D3034 D3046  ; #1腔体自检保压前真空值, #1腔体自检结果  0-未进行  1-自检中  2-自检OK  3-自检泄漏  4-自检抽真空NG
RSET W215.00  ; #1腔体抽真空失败
RSET W215.01  ; #1腔体自检结束
RSTA(531) W123 &7 &8
RSTA(531) W124 &1 &15
RSTA(531) W125 &0 &3
TIMX(550) 0160 &1  ; #1腔体自检数据初始化延时
; rung 7
LD P_On
OUT TR0
AND 1312.01  ; #1腔体氦检阀打开、合模
AND T0356  ; #1合模气缸缩回位延时
SET W211.08  ; #1合模气缸自检伸出
RSET W211.07  ; #1合模气缸自检缩回
LD TR0
AND 1312.01  ; #1腔体氦检阀打开、合模
AND T0468  ; #2氦检气缸原位延时
SET W215.08  ; #1腔体自检#2抽真空阀关闭
LD TR0
AND W61.07  ; #1合模气缸缩回位复位
RSET W211.08  ; #1合模气缸自检伸出

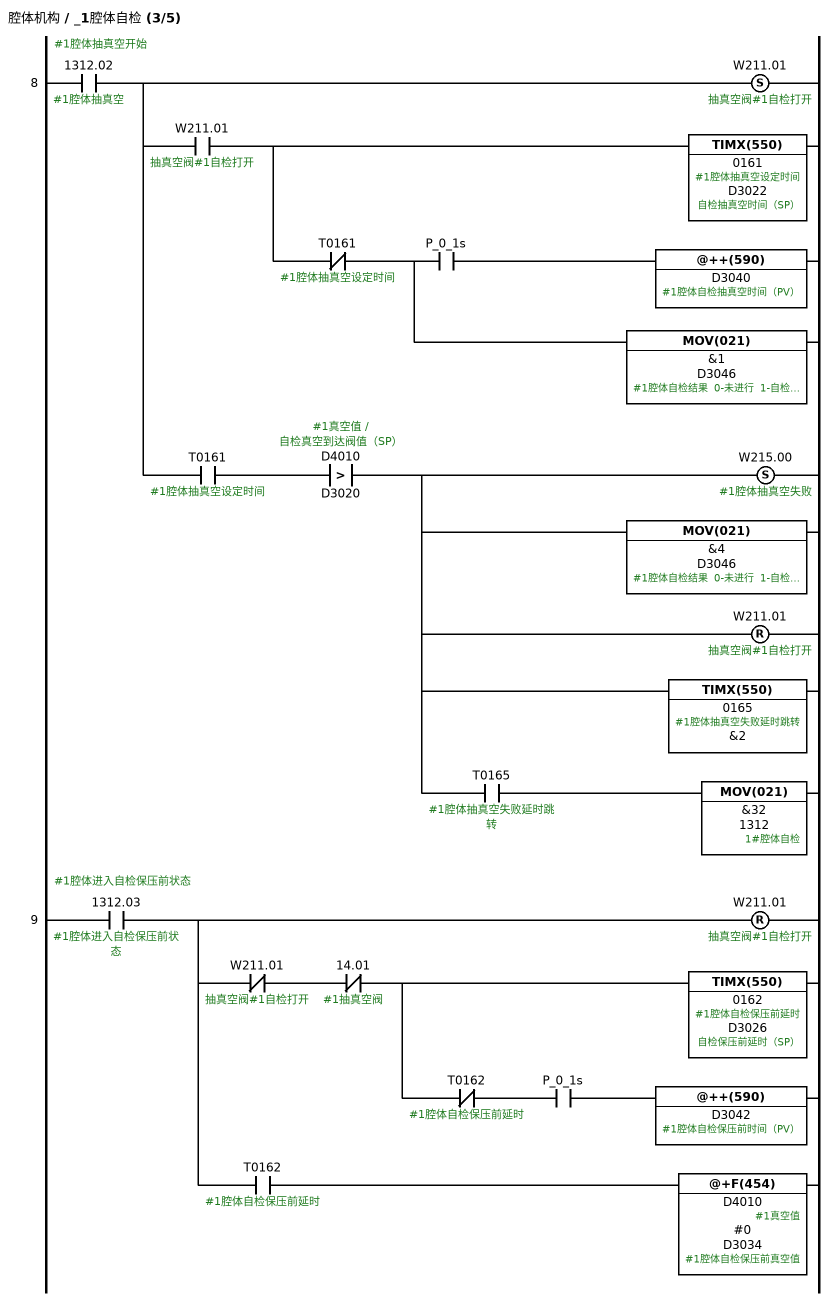
; rung 8: #1腔体抽真空开始
LD 1312.02  ; #1腔体抽真空
OUT TR0
SET W211.01  ; 抽真空阀#1自检打开
AND W211.01  ; 抽真空阀#1自检打开
TIMX(550) 0161 D3022  ; 自检抽真空时间（SP）, #1腔体抽真空设定时间
ANDNOT T0161  ; #1腔体抽真空设定时间
OUT TR1
AND P_0_1s
@++(590) D3040  ; #1腔体自检抽真空时间（PV）
LD TR1
MOV(021) &1 D3046  ; #1腔体自检结果  0-未进行  1-自检中  2-自检OK  3-自检泄漏  4-自检抽真空NG
LD TR0
AND T0161  ; #1腔体抽真空设定时间
AND>F(333) D4010 D3020  ; #1真空值, 自检真空到达阀值（SP）
SET W215.00  ; #1腔体抽真空失败
MOV(021) &4 D3046  ; #1腔体自检结果  0-未进行  1-自检中  2-自检OK  3-自检泄漏  4-自检抽真空NG
RSET W211.01  ; 抽真空阀#1自检打开
TIMX(550) 0165 &2  ; #1腔体抽真空失败延时跳转
AND T0165  ; #1腔体抽真空失败延时跳转
MOV(021) &32 1312  ; 1#腔体自检
; rung 9: #1腔体进入自检保压前状态
LD 1312.03  ; #1腔体进入自检保压前状态
OUT TR0
RSET W211.01  ; 抽真空阀#1自检打开
ANDNOT W211.01  ; 抽真空阀#1自检打开
ANDNOT 14.01  ; #1抽真空阀
TIMX(550) 0162 D3026  ; 自检保压前延时（SP）, #1腔体自检保压前延时
ANDNOT T0162  ; #1腔体自检保压前延时
AND P_0_1s
@++(590) D3042  ; #1腔体自检保压前时间（PV）
LD TR0
AND T0162  ; #1腔体自检保压前延时
@+F(454) D4010 #0 D3034  ; #1真空值, #1腔体自检保压前真空值

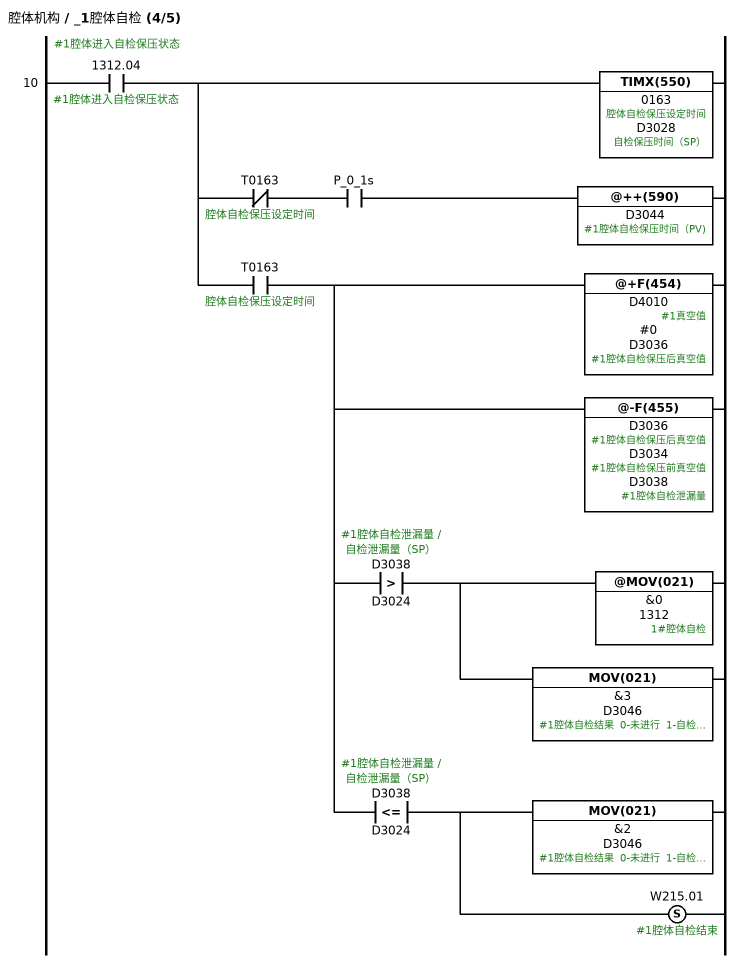
; rung 10: #1腔体进入自检保压状态
LD 1312.04  ; #1腔体进入自检保压状态
OUT TR0
TIMX(550) 0163 D3028  ; 自检保压时间（SP）, 腔体自检保压设定时间
ANDNOT T0163  ; 腔体自检保压设定时间
AND P_0_1s
@++(590) D3044  ; #1腔体自检保压时间（PV)
LD TR0
AND T0163  ; 腔体自检保压设定时间
OUT TR0
@+F(454) D4010 #0 D3036  ; #1真空值, #1腔体自检保压后真空值
@-F(455) D3036 D3034 D3038  ; #1腔体自检保压后真空值, #1腔体自检保压前真空值, #1腔体自检泄漏量
AND>F(333) D3038 D3024  ; #1腔体自检泄漏量, 自检泄漏量（SP）
@MOV(021) &0 1312  ; 1#腔体自检
MOV(021) &3 D3046  ; #1腔体自检结果  0-未进行  1-自检中  2-自检OK  3-自检泄漏  4-自检抽真空NG
LD TR0
AND<=F(332) D3038 D3024  ; #1腔体自检泄漏量, 自检泄漏量（SP）
MOV(021) &2 D3046  ; #1腔体自检结果  0-未进行  1-自检中  2-自检OK  3-自检泄漏  4-自检抽真空NG
SET W215.01  ; #1腔体自检结束

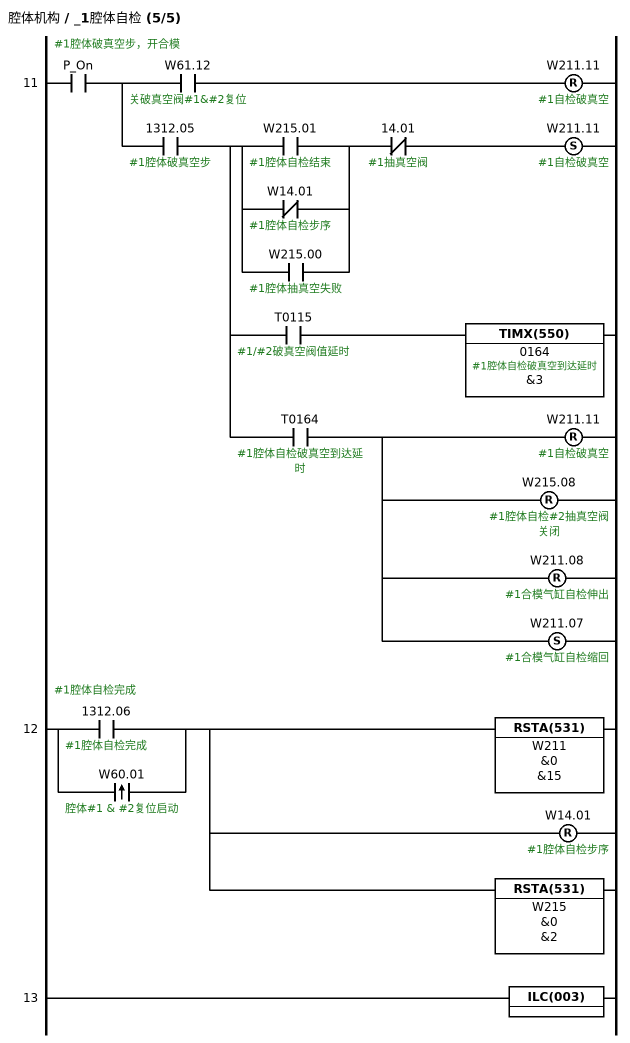
; rung 11: #1腔体破真空步，开合模
LD P_On
OUT TR0
AND W61.12  ; 关破真空阀#1&#2复位
RSET W211.11  ; #1自检破真空
LD TR0
AND 1312.05  ; #1腔体破真空步
OUT TR0
LD W215.01  ; #1腔体自检结束
ORNOT W14.01  ; #1腔体自检步序
OR W215.00  ; #1腔体抽真空失败
ANDLD
ANDNOT 14.01  ; #1抽真空阀
SET W211.11  ; #1自检破真空
LD TR0
AND T0115  ; #1/#2破真空阀值延时
TIMX(550) 0164 &3  ; #1腔体自检破真空到达延时
LD TR0
AND T0164  ; #1腔体自检破真空到达延时
RSET W211.11  ; #1自检破真空
RSET W215.08  ; #1腔体自检#2抽真空阀关闭
RSET W211.08  ; #1合模气缸自检伸出
SET W211.07  ; #1合模气缸自检缩回
; rung 12: #1腔体自检完成
LD 1312.06  ; #1腔体自检完成
@OR W60.01  ; 腔体#1 & #2复位启动
RSTA(531) W211 &0 &15
RSET W14.01  ; #1腔体自检步序
RSTA(531) W215 &0 &2
; rung 13
ILC(003)

### Section _2腔体自检

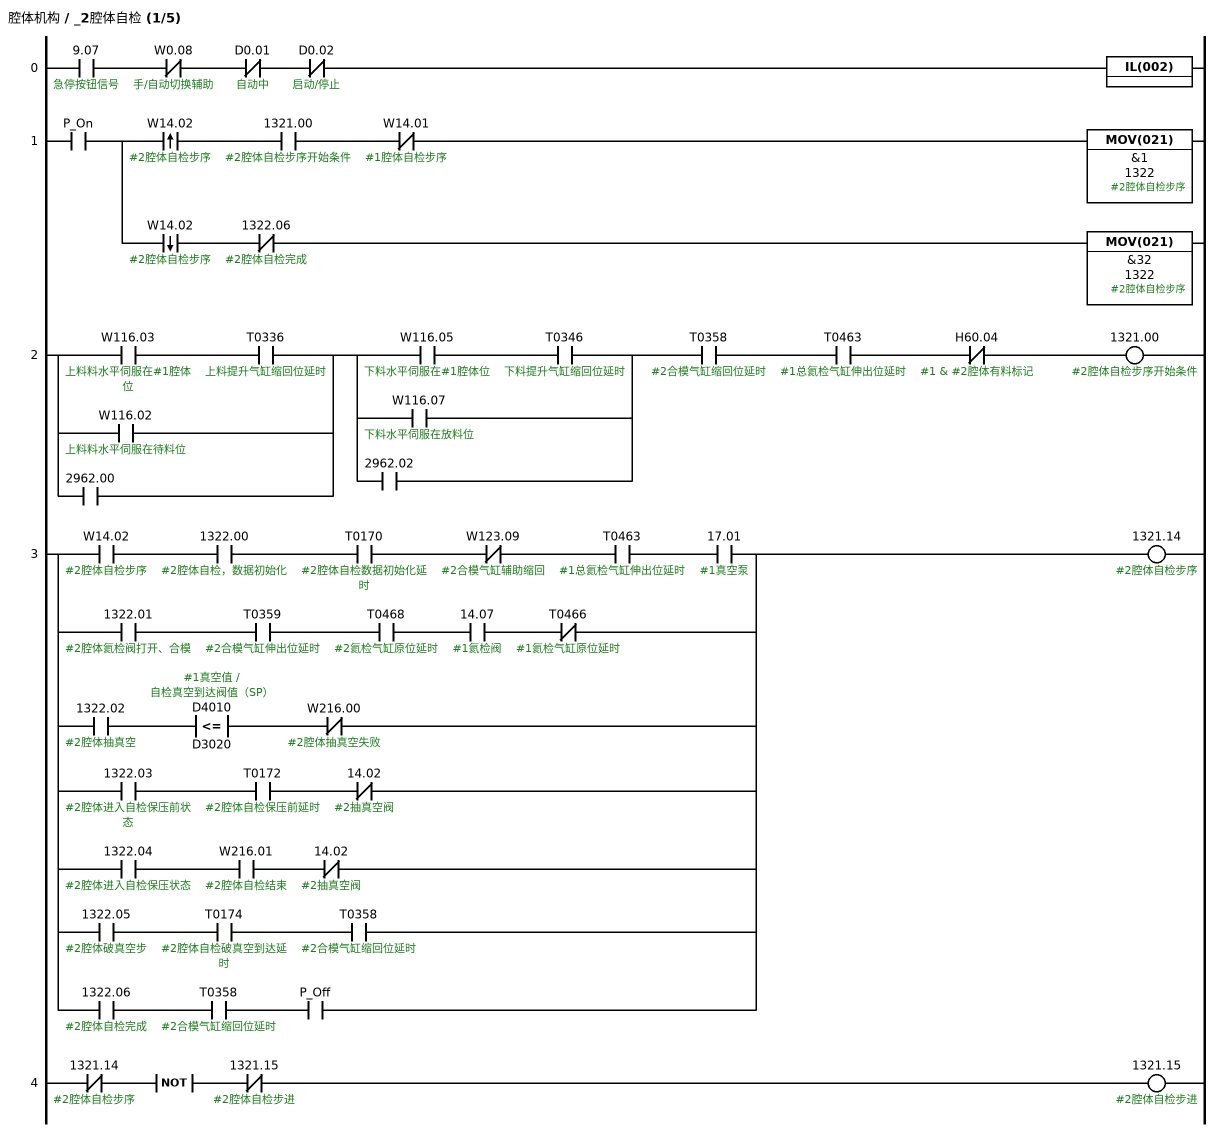
; rung 0
LD 9.07  ; 急停按钮信号
ANDNOT W0.08  ; 手/自动切换辅助
ANDNOT D0.01  ; 自动中
ANDNOT D0.02  ; 启动/停止
IL(002)
; rung 1
LD P_On
OUT TR0
@AND W14.02  ; #2腔体自检步序
AND 1321.00  ; #2腔体自检步序开始条件
ANDNOT W14.01  ; #1腔体自检步序
MOV(021) &1 1322  ; #2腔体自检步序
LD TR0
%AND W14.02  ; #2腔体自检步序
ANDNOT 1322.06  ; #2腔体自检完成
MOV(021) &32 1322  ; #2腔体自检步序
; rung 2
LD W116.03  ; 上料料水平伺服在#1腔体位
AND T0336  ; 上料提升气缸缩回位延时
OR W116.02  ; 上料料水平伺服在待料位
OR 2962.00
LD W116.05  ; 下料水平伺服在#1腔体位
AND T0346  ; 下料提升气缸缩回位延时
OR W116.07  ; 下料水平伺服在放料位
OR 2962.02
ANDLD
AND T0358  ; #2合模气缸缩回位延时
AND T0463  ; #1总氦检气缸伸出位延时
ANDNOT H60.04  ; #1 & #2腔体有料标记
OUT 1321.00  ; #2腔体自检步序开始条件
; rung 3
LD W14.02  ; #2腔体自检步序
AND 1322.00  ; #2腔体自检，数据初始化
AND T0170  ; #2腔体自检数据初始化延时
ANDNOT W123.09  ; #2合模气缸辅助缩回
AND T0463  ; #1总氦检气缸伸出位延时
AND 17.01  ; #1真空泵
LD 1322.01  ; #2腔体氦检阀打开、合模
AND T0359  ; #2合模气缸伸出位延时
AND T0468  ; #2氦检气缸原位延时
AND 14.07  ; #1氦检阀
ANDNOT T0466  ; #1氦检气缸原位延时
ORLD
LD 1322.02  ; #2腔体抽真空
AND<=F(332) D4010 D3020  ; #1真空值, 自检真空到达阀值（SP）
ANDNOT W216.00  ; #2腔体抽真空失败
ORLD
LD 1322.03  ; #2腔体进入自检保压前状态
AND T0172  ; #2腔体自检保压前延时
ANDNOT 14.02  ; #2抽真空阀
ORLD
LD 1322.04  ; #2腔体进入自检保压状态
AND W216.01  ; #2腔体自检结束
ANDNOT 14.02  ; #2抽真空阀
ORLD
LD 1322.05  ; #2腔体破真空步
AND T0174  ; #2腔体自检破真空到达延时
AND T0358  ; #2合模气缸缩回位延时
ORLD
LD 1322.06  ; #2腔体自检完成
AND T0358  ; #2合模气缸缩回位延时
AND P_Off
ORLD
OUT 1321.14  ; #2腔体自检步序
; rung 4
LDNOT 1321.14  ; #2腔体自检步序
NOT(520)
ANDNOT 1321.15  ; #2腔体自检步进
OUT 1321.15  ; #2腔体自检步进

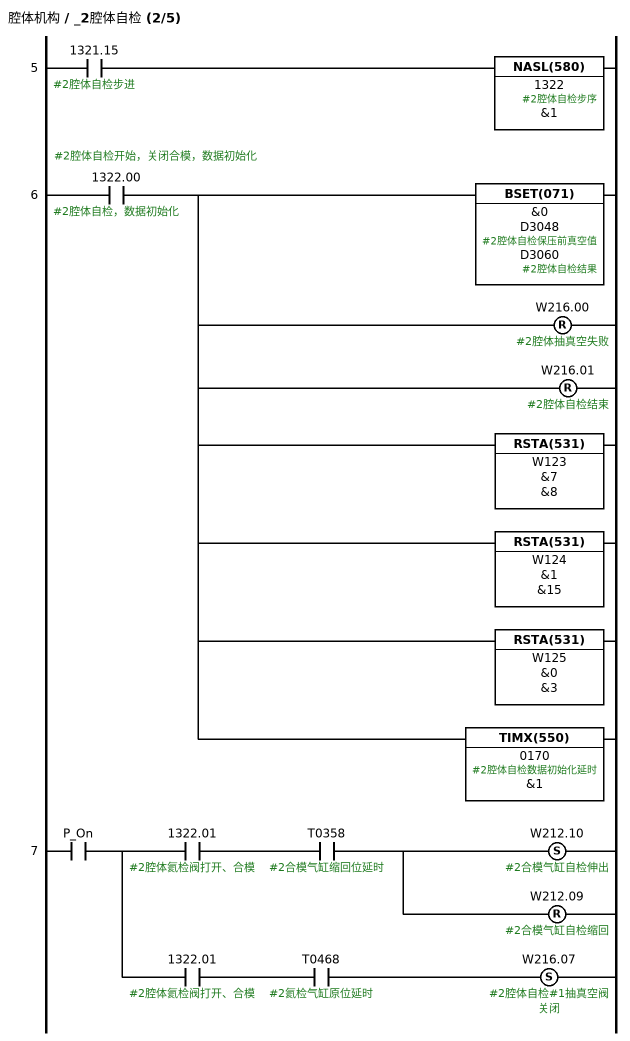
; rung 5
LD 1321.15  ; #2腔体自检步进
NASL(580) 1322 &1  ; #2腔体自检步序
; rung 6: #2腔体自检开始，关闭合模，数据初始化
LD 1322.00  ; #2腔体自检，数据初始化
BSET(071) &0 D3048 D3060  ; #2腔体自检保压前真空值, #2腔体自检结果
RSET W216.00  ; #2腔体抽真空失败
RSET W216.01  ; #2腔体自检结束
RSTA(531) W123 &7 &8
RSTA(531) W124 &1 &15
RSTA(531) W125 &0 &3
TIMX(550) 0170 &1  ; #2腔体自检数据初始化延时
; rung 7
LD P_On
OUT TR0
AND 1322.01  ; #2腔体氦检阀打开、合模
AND T0358  ; #2合模气缸缩回位延时
SET W212.10  ; #2合模气缸自检伸出
RSET W212.09  ; #2合模气缸自检缩回
LD TR0
AND 1322.01  ; #2腔体氦检阀打开、合模
AND T0468  ; #2氦检气缸原位延时
SET W216.07  ; #2腔体自检#1抽真空阀关闭

